// TIA Portal project "KananBagaliyev_Project" (V14)

(* hardware
DEVICE "S7300/ET200M station_1"  S7-300 station
   slot 0: "Rail_0"  Rail  6ES7 390-1***0-0AA0
   slot 1: "PS 307 10A_1"  PS 307 10A  6ES7 307-1KA02-0AA0
   slot 2: "PLC_1"  CPU 315-2 PN/DP  6ES7 315-2EH14-0AB0  V3.2
      slot 2: "PROFINET interface_1"  PN-IO
         slot 1: "Port_1"  Port
         slot 2: "Port_2"  Port
   slot 4: "DI 16x24VDC_1"  DI16 x 24VDC  6ES7 321-1BH50-0AA0
   slot 5: "DO 16x24VDC/0.5A_1"  DO16xDC24V/0.5A  6ES7 322-8BH10-0AB0
   slot 6: "AI 8x16BIT_1"  AI8 x 16 bits  6ES7 331-7NF10-0AB0
DEVICE "PC-System_1"  SIMATIC PC station
   slot 0: "SIMATIC PC station"  Rail  SIMATIC PC-Station  V1.0
      slot 125: "Stationmanager"  Station_Manager  V6.0.4
   slot 1: "HMI_RT_1"  WinCC RT Advanced  6AV2 104-0xxxx-xxxx  14.0.0.0
      slot 33792: "Host interface"  Host interface
   slot 2: "IE general_1"  IE General  IE_CP  V8.2.0
*)

// ===== PLC "PLC_1"  CPU 315-2 PN/DP =====

VAR_GLOBAL   // PLC tag table "Default tag table"
   "LT1401" AT %MW288 : Int;
   "LT1501" AT %MW290 : Int;
   "LT1601" AT %MW292 : Int;
   "LT1701" AT %MW294 : Int;
   "Pump100A_start" AT %M0.0 : Bool;
   "Pump100A_stop" AT %M0.1 : Bool;
   "Pump770A_start" AT %M0.2 : Bool;
   "Pump770A_stop" AT %M0.3 : Bool;
   "Pump771A_start" AT %M0.4 : Bool;
   "Pump771A_stop" AT %M0.5 : Bool;
   "Pump100A" AT %Q4.0 : Bool;
   "Pump770A" AT %Q4.1 : Bool;
   "Pump771A" AT %Q4.2 : Bool;
   "SV1401" AT %Q4.3 : Bool;
   "SV1402" AT %Q4.4 : Bool;
   "SV1501" AT %Q4.5 : Bool;
   "SV1502" AT %Q4.6 : Bool;
   "SV1601" AT %Q4.7 : Bool;
   "SV1602" AT %Q5.0 : Bool;
   "SV1701" AT %Q5.1 : Bool;
   "SV1702" AT %Q5.2 : Bool;
   "SV1401_open" AT %M0.6 : Bool;
   "SV1401_close" AT %M0.7 : Bool;
   "SV1402_open" AT %M1.0 : Bool;
   "SV1402_close" AT %M1.1 : Bool;
   "SV1501_open" AT %M1.2 : Bool;
   "SV1501_close" AT %M1.3 : Bool;
   "SV1502_open" AT %M1.4 : Bool;
   "SV1502_close" AT %M1.5 : Bool;
   "SV1601_open" AT %M1.6 : Bool;
   "SV1601_close" AT %M1.7 : Bool;
   "SV1602_open" AT %M2.0 : Bool;
   "SV1602_close" AT %M2.1 : Bool;
   "SV1701_open" AT %M2.2 : Bool;
   "SV1701_close" AT %M2.3 : Bool;
   "SV1702_open" AT %M2.4 : Bool;
   "SV1702_close" AT %M2.5 : Bool;
   "140L" AT %M2.6 : Bool;
   "140LL" AT %M2.7 : Bool;
   "140H" AT %M3.0 : Bool;
   "140HH" AT %M3.1 : Bool;
   "150L" AT %M3.2 : Bool;
   "150LL" AT %M3.3 : Bool;
   "150H" AT %M3.4 : Bool;
   "150HH" AT %M3.5 : Bool;
   "160L" AT %M3.6 : Bool;
   "160LL" AT %M3.7 : Bool;
   "160H" AT %M4.0 : Bool;
   "160HH" AT %M4.1 : Bool;
   "170L" AT %M4.2 : Bool;
   "170LL" AT %M4.3 : Bool;
   "170H" AT %M4.4 : Bool;
   "170HH" AT %M4.5 : Bool;
   "140_real" AT %MD200 : Real;
   "150_real" AT %MD204 : Real;
   "160_real" AT %MD208 : Real;
   "170_real" AT %MD212 : Real;
END_VAR

VAR_GLOBAL CONSTANT   // PLC tag table "Default tag table"
   "140L_SP" : Real := 150.0;
   "140LL_SP" : Real := 75.0;
   "140H_SP" : Real := 1350.0;
   "140HH_SP" : Real := 1425.0;
   "150L_SP" : Real := 250.0;
   "150LL_SP" : Real := 125.0;
   "150H_SP" : Real := 2250.0;
   "150HH_SP" : Real := 2375.0;
   "160L_SP" : Real := 300.0;
   "160LL_SP" : Real := 150.0;
   "160H_SP" : Real := 2700.0;
   "160HH_SP" : Real := 2850.0;
   "170L_SP" : Real := 1000.0;
   "170LL_SP" : Real := 500.0;
   "170H_SP" : Real := 9000.0;
   "170HH_SP" : Real := 9500.0;
   "140_capacity_max" : Real := 1500.0;
   "150_capacity_max" : Real := 2500.0;
   "160_capacity_max" : Real := 3000.0;
   "170_capacity_max" : Real := 10000.0;
   "140_capacity_min" : Real := 0.0;
   "150_capacity_min" : Real := 0.0;
   "160_capacity_min" : Real := 0.0;
   "170_capacity_min" : Real := 0.0;
END_VAR

DATA_BLOCK "FP_DB"   // DB1
{ S7_Optimized_Access := 'FALSE' }
VERSION : 0.1
   VAR
      FP_visibility_PUMP_100A : Bool := false;
      FP_visibility_PUMP_770A : Bool := false;
      FP_visibility_PUMP_771A : Bool := false;
      FP_tag_number_PUMP_100A : String := 'PUMP_100_A';
      FP_tag_number_PUMP_770A : String := 'PUMP_770_A';
      FP_tag_number_PUMP_771A : String := 'PUMP_771_A';
      FP_visibility_SV1401 : Bool := false;
      FP_visibility_SV1402 : Bool := false;
      FP_visibility_SV1501 : Bool := false;
      FP_visibility_SV1502 : Bool := false;
      FP_visibility_SV1601 : Bool := false;
      FP_visibility_SV1602 : Bool := false;
      FP_visibility_SV1701 : Bool := false;
      FP_visibility_SV1702 : Bool := false;
      FP_tag_number_SV1401 : String := 'SV1401';
      FP_tag_number_SV1402 : String := 'SV1402';
      FP_tag_number_SV1501 : String := 'SV1501';
      FP_tag_number_SV1502 : String := 'SV1502';
      FP_tag_number_SV1601 : String := 'SV1601';
      FP_tag_number_SV1602 : String := 'SV1602';
      FP_tag_number_SV1701 : String := 'SV1701';
      FP_tag_number_SV1702 : String := 'SV1702';
   END_VAR
BEGIN
END_DATA_BLOCK

DATA_BLOCK "Tank140Fill_DB"   // DB2
{ S7_Optimized_Access := 'FALSE' }
VERSION : 0.1
// stored: InstanceOfName FillTank
"FillTank"
BEGIN
END_DATA_BLOCK

DATA_BLOCK "Tank150Fill_DB"   // DB3
{ S7_Optimized_Access := 'FALSE' }
VERSION : 0.1
// stored: InstanceOfName FillTank
"FillTank"
BEGIN
END_DATA_BLOCK

DATA_BLOCK "Tank160Fill_DB"   // DB4
{ S7_Optimized_Access := 'FALSE' }
VERSION : 0.1
// stored: InstanceOfName FillTank
"FillTank"
BEGIN
END_DATA_BLOCK

DATA_BLOCK "DrainMasterTank_DB"   // DB5
{ S7_Optimized_Access := 'FALSE' }
VERSION : 0.1
// stored: InstanceOfName DrainMasterTank
"DrainMasterTank"
BEGIN
END_DATA_BLOCK

FUNCTION_BLOCK "FillTank"   // FB1, LAD
{ S7_Optimized_Access := 'FALSE' }
VERSION : 0.1
   VAR_INPUT
      SV1x02 : Bool;
      SV1x01 : Bool;
      Pump : Bool;
      Reduction_rate : Int;
   END_VAR
   VAR_IN_OUT
      LT1x01 : Int;
   END_VAR
   VAR
      "timer" : Time;
      IEC_Timer_0_Instance : TON;
      IEC_Timer_0_Instance_1 : TON;
      timer_1 : Time;
   END_VAR
BEGIN

REGION Network 1: Fill Tank timer
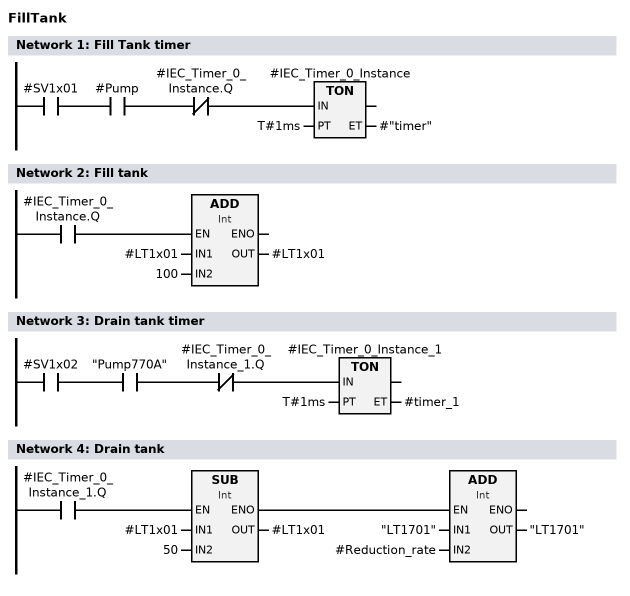
   #IEC_Timer_0_Instance.TON(IN := #SV1x01 AND #Pump AND NOT #IEC_Timer_0_Instance.Q,
                           PT := T#1ms,
                           ET => #"timer");
END_REGION

REGION Network 2: Fill tank
   RUNG wire#powerrail
      Contact( #IEC_Timer_0_Instance.Q )
      { S7_Templates := "SrcType := Int"; S7_GenerateENO := "TRUE" } Add(in1 := #LT1x01, in2 := 100, out => #LT1x01)
   END_RUNG
   // the same network as SCL:
   IF #IEC_Timer_0_Instance.Q THEN #LT1x01 := #LT1x01 + 100; END_IF;
END_REGION

REGION Network 3: Drain tank timer
   #IEC_Timer_0_Instance_1.TON(IN := #SV1x02 AND "Pump770A" AND NOT #IEC_Timer_0_Instance_1.Q,
                           PT := T#1ms,
                           ET => #timer_1);
END_REGION

REGION Network 4: Drain tank
   RUNG wire#powerrail
      Contact( #IEC_Timer_0_Instance_1.Q )
      { S7_Templates := "SrcType := Int"; S7_GenerateENO := "TRUE" } Sub(in1 := #LT1x01, in2 := 50, out => #LT1x01)
      { S7_Templates := "SrcType := Int"; S7_GenerateENO := "TRUE" } Add(in1 := "LT1701", in2 := #Reduction_rate, out => "LT1701")
   END_RUNG
   // the same network as SCL:
   // ENO of a box is taken as its EN; it also drops when the box reports an error
   IF #IEC_Timer_0_Instance_1.Q THEN
       #LT1x01 := #LT1x01 - 50;
       "LT1701" := "LT1701" + #Reduction_rate;
   END_IF;
END_REGION
END_FUNCTION_BLOCK

FUNCTION_BLOCK "DrainMasterTank"   // FB2, LAD
{ S7_Optimized_Access := 'FALSE' }
VERSION : 0.1
   VAR
      IEC_Timer_0_Instance : TON;
      "timer" : Time;
   END_VAR
BEGIN

REGION Network 1
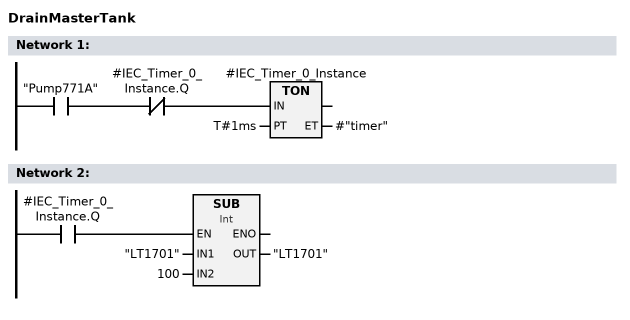
   #IEC_Timer_0_Instance.TON(IN := "Pump771A" AND NOT #IEC_Timer_0_Instance.Q, PT := T#1ms, ET => #"timer");
END_REGION

REGION Network 2
   RUNG wire#powerrail
      Contact( #IEC_Timer_0_Instance.Q )
      { S7_Templates := "SrcType := Int"; S7_GenerateENO := "TRUE" } Sub(in1 := "LT1701", in2 := 100, out => "LT1701")
   END_RUNG
   // the same network as SCL:
   IF #IEC_Timer_0_Instance.Q THEN "LT1701" := "LT1701" - 100; END_IF;
END_REGION
END_FUNCTION_BLOCK

FUNCTION "TankAlarm" : Void   // FC1, LAD
{ S7_Optimized_Access := 'FALSE' }
VERSION : 0.1
   VAR_INPUT
      LT1x01 : Int;
      max_level : Real;
      min_level : Real;
      high_alarm_sp : Real;
      low_alarm_sp : Real;
      hh_alarm_sp : Real;
      ll_alarm_sp : Real;
   END_VAR
   VAR_OUTPUT
      high_alarm : Bool;
      low_alarm : Bool;
      hh_alarm : Bool;
      ll_alarm : Bool;
   END_VAR
   VAR_IN_OUT
      level_real : Real;
   END_VAR
   VAR_TEMP
      bipolar : Bool;
      value : Word;
   END_VAR
BEGIN

REGION Network 1
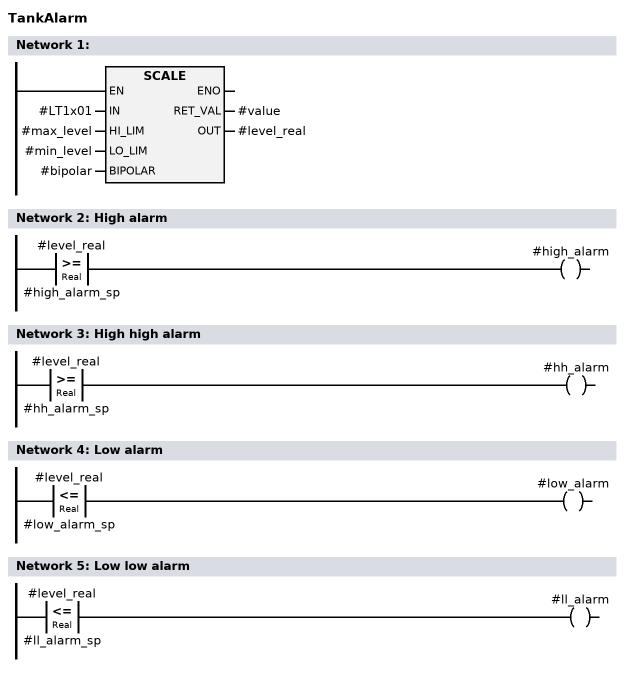
   #value := SCALE(IN := #LT1x01,
                   HI_LIM := #max_level,
                   LO_LIM := #min_level,
                   BIPOLAR := #bipolar,
                   OUT => #level_real);
END_REGION

REGION Network 2: High alarm
   RUNG wire#powerrail
      { S7_Templates := "SrcType := Real" } GE_Contact(in1 := #level_real, in2 := #high_alarm_sp)
      Coil( #high_alarm )
   END_RUNG
   // the same network as SCL:
   #high_alarm := #level_real >= #high_alarm_sp;
END_REGION

REGION Network 3: High high alarm
   RUNG wire#powerrail
      { S7_Templates := "SrcType := Real" } GE_Contact(in1 := #level_real, in2 := #hh_alarm_sp)
      Coil( #hh_alarm )
   END_RUNG
   // the same network as SCL:
   #hh_alarm := #level_real >= #hh_alarm_sp;
END_REGION

REGION Network 4: Low alarm
   RUNG wire#powerrail
      { S7_Templates := "SrcType := Real" } LE_Contact(in1 := #level_real, in2 := #low_alarm_sp)
      Coil( #low_alarm )
   END_RUNG
   // the same network as SCL:
   #low_alarm := #level_real <= #low_alarm_sp;
END_REGION

REGION Network 5: Low low alarm
   RUNG wire#powerrail
      { S7_Templates := "SrcType := Real" } LE_Contact(in1 := #level_real, in2 := #ll_alarm_sp)
      Coil( #ll_alarm )
   END_RUNG
   // the same network as SCL:
   #ll_alarm := #level_real <= #ll_alarm_sp;
END_REGION
END_FUNCTION

FUNCTION "SV1x01" : Void   // FC2, LAD
{ S7_Optimized_Access := 'FALSE' }
VERSION : 0.1
   VAR_INPUT
      Open_valve : Bool;
      Close_valve : Bool;
      HH_alarm : Bool;
      Inlet_pump_stop : Bool;
   END_VAR
   VAR_OUTPUT
      SV1x01 : Bool;
   END_VAR
BEGIN

REGION Network 1
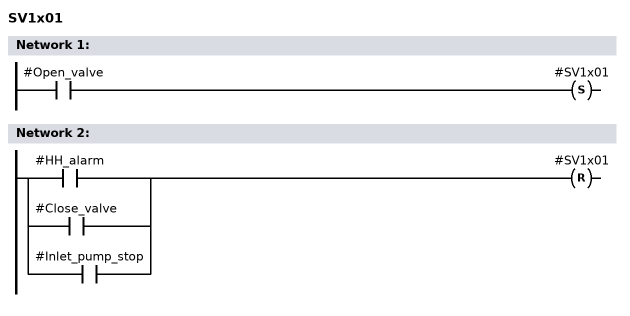
   RUNG wire#powerrail
      Contact( #Open_valve )
      S_Coil( #SV1x01 )
   END_RUNG
   // the same network as SCL:
   IF #Open_valve THEN #SV1x01 := TRUE; END_IF;
END_REGION

REGION Network 2
   RUNG wire#powerrail
      Contact( #HH_alarm )
      wire#w1
      R_Coil( #SV1x01 )
   END_RUNG
   RUNG wire#powerrail
      Contact( #Close_valve )
   END_RUNG wire#w1
   RUNG wire#powerrail
      Contact( #Inlet_pump_stop )
   END_RUNG wire#w1
   // the same network as SCL:
   IF #HH_alarm OR #Close_valve OR #Inlet_pump_stop THEN #SV1x01 := FALSE; END_IF;
END_REGION
END_FUNCTION

FUNCTION "Pump_100A" : Void   // FC3, LAD
{ S7_Optimized_Access := 'FALSE' }
VERSION : 0.1
   VAR_INPUT
      SV1x01_1 : Bool;
      SV1x01_2 : Bool;
      SV1x01_3 : Bool;
      Start_pump : Bool;
      Stop_pump : Bool;
   END_VAR
   VAR_OUTPUT
      Pump100A : Bool;
   END_VAR
BEGIN

REGION Network 1
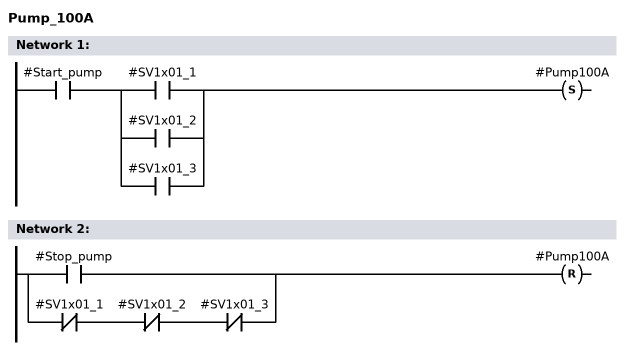
   RUNG wire#powerrail
      Contact( #Start_pump )
      wire#w1
      Contact( #SV1x01_1 )
      wire#w2
      S_Coil( #Pump100A )
   END_RUNG
   RUNG wire#w1
      Contact( #SV1x01_2 )
   END_RUNG wire#w2
   RUNG wire#w1
      Contact( #SV1x01_3 )
   END_RUNG wire#w2
   // the same network as SCL:
   IF #Start_pump AND (#SV1x01_1 OR #SV1x01_2 OR #SV1x01_3) THEN #Pump100A := TRUE; END_IF;
END_REGION

REGION Network 2
   RUNG wire#powerrail
      Contact( #Stop_pump )
      wire#w1
      R_Coil( #Pump100A )
   END_RUNG
   RUNG wire#powerrail
      I_Contact( #SV1x01_1 )
      I_Contact( #SV1x01_2 )
      I_Contact( #SV1x01_3 )
   END_RUNG wire#w1
   // the same network as SCL:
   IF #Stop_pump OR (NOT #SV1x01_1 AND NOT #SV1x01_2 AND NOT #SV1x01_3) THEN #Pump100A := FALSE; END_IF;
END_REGION
END_FUNCTION

FUNCTION "SV1x02_slaves" : Void   // FC4, LAD
{ S7_Optimized_Access := 'FALSE' }
VERSION : 0.1
   VAR_INPUT
      Valve_open : Bool;
      Valve_close : Bool;
      "170L" : Bool;
      "1x0L" : Bool;
      Pump_770_A_stop : Bool;
      "170H" : Bool;
   END_VAR
   VAR_OUTPUT
      Valve_energize : Bool;
   END_VAR
BEGIN

REGION Network 1
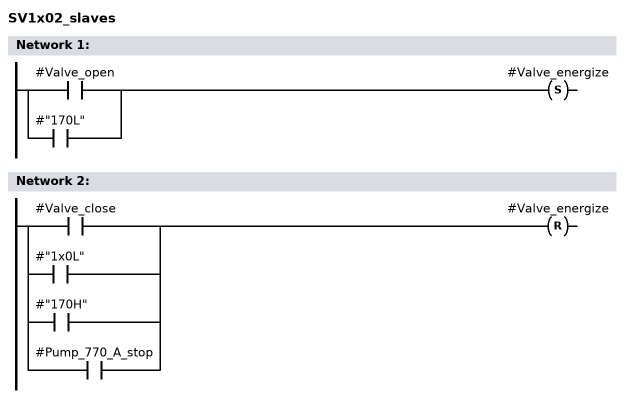
   RUNG wire#powerrail
      Contact( #Valve_open )
      wire#w1
      S_Coil( #Valve_energize )
   END_RUNG
   RUNG wire#powerrail
      Contact( #"170L" )
   END_RUNG wire#w1
   // the same network as SCL:
   IF #Valve_open OR #"170L" THEN #Valve_energize := TRUE; END_IF;
END_REGION

REGION Network 2
   RUNG wire#powerrail
      Contact( #Valve_close )
      wire#w1
      R_Coil( #Valve_energize )
   END_RUNG
   RUNG wire#powerrail
      Contact( #"1x0L" )
   END_RUNG wire#w1
   RUNG wire#powerrail
      Contact( #"170H" )
   END_RUNG wire#w1
   RUNG wire#powerrail
      Contact( #Pump_770_A_stop )
   END_RUNG wire#w1
   // the same network as SCL:
   IF #Valve_close OR #"1x0L" OR #"170H" OR #Pump_770_A_stop THEN #Valve_energize := FALSE; END_IF;
END_REGION
END_FUNCTION

FUNCTION "SV_1702" : Void   // FC5, LAD
{ S7_Optimized_Access := 'FALSE' }
VERSION : 0.1
   VAR_INPUT
      Valve_open : Bool;
      Valve_close : Bool;
      "170L" : Bool;
      Pump_771_A : Bool;
   END_VAR
   VAR_OUTPUT
      Valve_energize : Bool;
   END_VAR
BEGIN

REGION Network 1
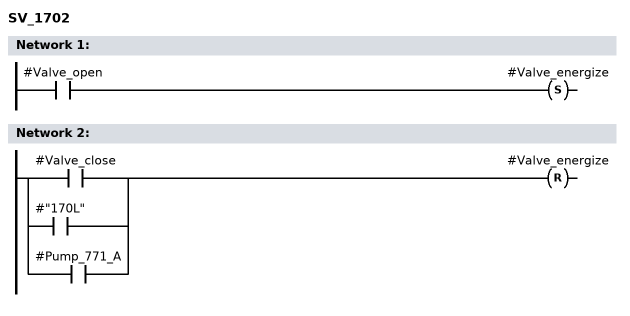
   RUNG wire#powerrail
      Contact( #Valve_open )
      S_Coil( #Valve_energize )
   END_RUNG
   // the same network as SCL:
   IF #Valve_open THEN #Valve_energize := TRUE; END_IF;
END_REGION

REGION Network 2
   RUNG wire#powerrail
      Contact( #Valve_close )
      wire#w1
      R_Coil( #Valve_energize )
   END_RUNG
   RUNG wire#powerrail
      Contact( #"170L" )
   END_RUNG wire#w1
   RUNG wire#powerrail
      Contact( #Pump_771_A )
   END_RUNG wire#w1
   // the same network as SCL:
   IF #Valve_close OR #"170L" OR #Pump_771_A THEN #Valve_energize := FALSE; END_IF;
END_REGION
END_FUNCTION

FUNCTION "Pump_770A" : Void   // FC6, LAD
{ S7_Optimized_Access := 'FALSE' }
VERSION : 0.1
   VAR_INPUT
      Start_pump : Bool;
      Stop_pump : Bool;
      SV1701 : Bool;
      SV1402 : Bool;
      SV1502 : Bool;
      SV1602 : Bool;
      "170L" : Bool;
      "170H" : Bool;
   END_VAR
   VAR_OUTPUT
      Pump_770A : Bool;
   END_VAR
BEGIN

REGION Network 1
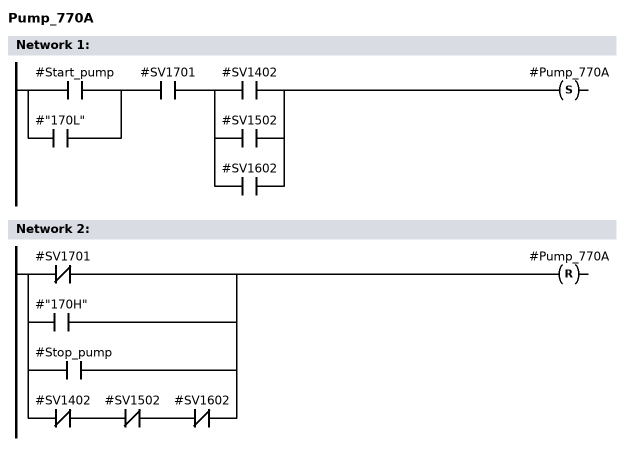
   RUNG wire#powerrail
      Contact( #Start_pump )
      wire#w1
      Contact( #SV1701 )
      wire#w2
      Contact( #SV1402 )
      wire#w3
      S_Coil( #Pump_770A )
   END_RUNG
   RUNG wire#powerrail
      Contact( #"170L" )
   END_RUNG wire#w1
   RUNG wire#w2
      Contact( #SV1502 )
   END_RUNG wire#w3
   RUNG wire#w2
      Contact( #SV1602 )
   END_RUNG wire#w3
   // the same network as SCL:
   IF (#Start_pump OR #"170L") AND #SV1701 AND (#SV1402 OR #SV1502 OR #SV1602) THEN
       #Pump_770A := TRUE;
   END_IF;
END_REGION

REGION Network 2
   RUNG wire#powerrail
      I_Contact( #SV1701 )
      wire#w1
      R_Coil( #Pump_770A )
   END_RUNG
   RUNG wire#powerrail
      Contact( #"170H" )
   END_RUNG wire#w1
   RUNG wire#powerrail
      Contact( #Stop_pump )
   END_RUNG wire#w1
   RUNG wire#powerrail
      I_Contact( #SV1402 )
      I_Contact( #SV1502 )
      I_Contact( #SV1602 )
   END_RUNG wire#w1
   // the same network as SCL:
   IF NOT #SV1701 OR #"170H" OR #Stop_pump OR (NOT #SV1402 AND NOT #SV1502 AND NOT #SV1602) THEN
       #Pump_770A := FALSE;
   END_IF;
END_REGION
END_FUNCTION

FUNCTION "Pump_771A" : Void   // FC7, LAD
{ S7_Optimized_Access := 'FALSE' }
VERSION : 0.1
   VAR_INPUT
      Pump_start : Bool;
      SV1702 : Bool;
      Pump_stop : Bool;
      "170L" : Bool;
   END_VAR
   VAR_OUTPUT
      Pump_771A : Bool;
   END_VAR
BEGIN

REGION Network 1
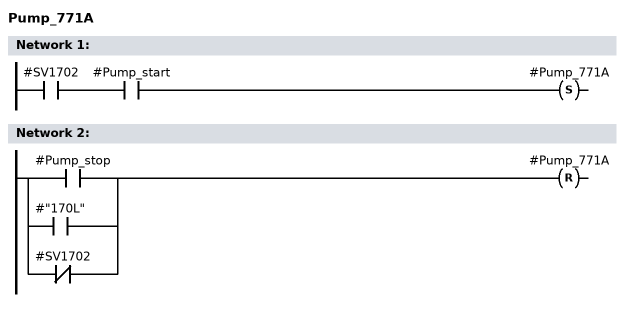
   RUNG wire#powerrail
      Contact( #SV1702 )
      Contact( #Pump_start )
      S_Coil( #Pump_771A )
   END_RUNG
   // the same network as SCL:
   IF #SV1702 AND #Pump_start THEN #Pump_771A := TRUE; END_IF;
END_REGION

REGION Network 2
   RUNG wire#powerrail
      Contact( #Pump_stop )
      wire#w1
      R_Coil( #Pump_771A )
   END_RUNG
   RUNG wire#powerrail
      Contact( #"170L" )
   END_RUNG wire#w1
   RUNG wire#powerrail
      I_Contact( #SV1702 )
   END_RUNG wire#w1
   // the same network as SCL:
   IF #Pump_stop OR #"170L" OR NOT #SV1702 THEN #Pump_771A := FALSE; END_IF;
END_REGION
END_FUNCTION

ORGANIZATION_BLOCK "Main"   // OB1, LAD
TITLE = "Main Program Sweep (Cycle)"
{ S7_Optimized_Access := 'FALSE' }
VERSION : 0.1
   VAR_TEMP
      OB1_EV_CLASS : Byte;   // Bits 0-3 = 1 (Coming event), Bits 4-7 = 1 (Event class 1)
      OB1_SCAN_1 : Byte;   // 1 (Cold restart scan 1 of OB 1), 3 (Scan 2-n of OB 1)
      OB1_PRIORITY : Byte;   // Priority of OB Execution
      OB1_OB_NUMBR : Byte;   // 1 (Organization block 1, OB1)
      OB1_RESERVED_1 : Byte;   // Reserved for system
      OB1_RESERVED_2 : Byte;   // Reserved for system
      OB1_PREV_CYCLE : Int;   // Cycle time of previous OB1 scan (milliseconds)
      OB1_MIN_CYCLE : Int;   // Minimum cycle time of OB1 (milliseconds)
      OB1_MAX_CYCLE : Int;   // Maximum cycle time of OB1 (milliseconds)
      OB1_DATE_TIME : Date_And_Time;   // Date and time OB1 started
   END_VAR
BEGIN

REGION Network 1: Tank 140
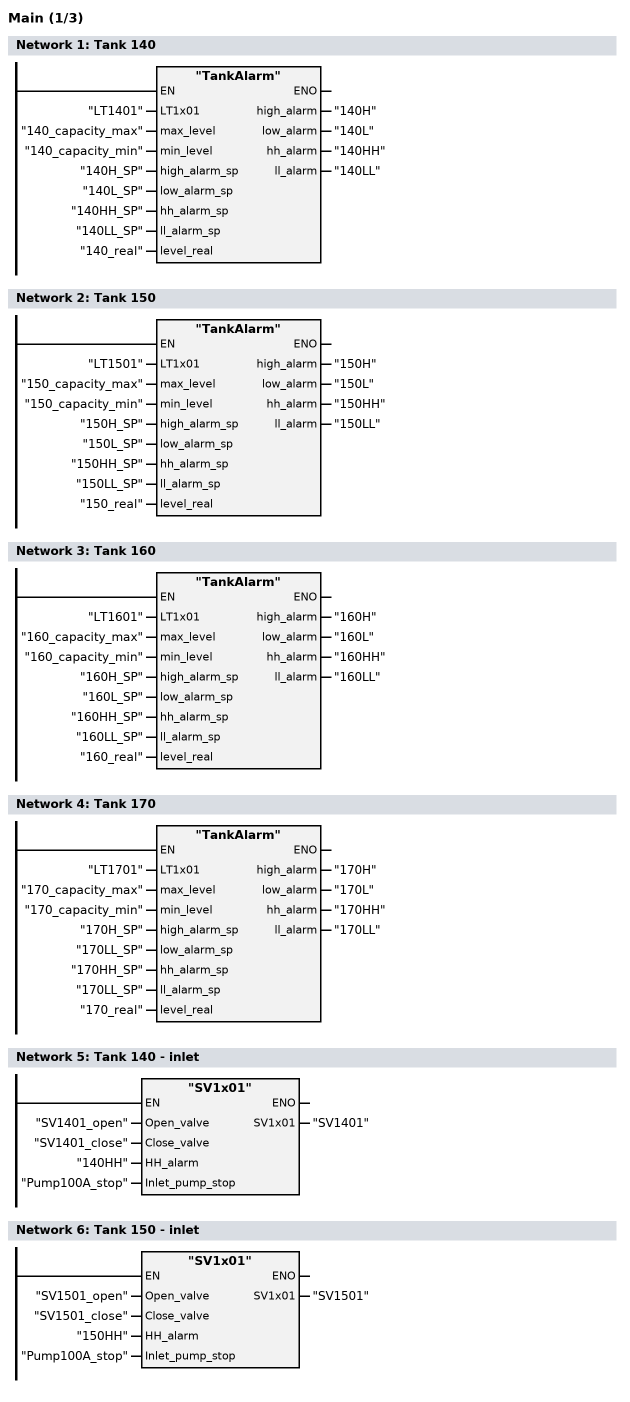
   RUNG wire#powerrail
      "TankAlarm"(LT1x01 := "LT1401", max_level := "140_capacity_max", min_level := "140_capacity_min", high_alarm_sp := "140H_SP", low_alarm_sp := "140L_SP", hh_alarm_sp := "140HH_SP", ll_alarm_sp := "140LL_SP", level_real := "140_real", high_alarm => "140H", low_alarm => "140L", hh_alarm => "140HH", ll_alarm => "140LL")
   END_RUNG
   // the same network as SCL:
   "TankAlarm"(LT1x01 := "LT1401",
               max_level := "140_capacity_max",
               min_level := "140_capacity_min",
               high_alarm_sp := "140H_SP",
               low_alarm_sp := "140L_SP",
               hh_alarm_sp := "140HH_SP",
               ll_alarm_sp := "140LL_SP",
               level_real := "140_real",
               high_alarm => "140H",
               low_alarm => "140L",
               hh_alarm => "140HH",
               ll_alarm => "140LL");
END_REGION

REGION Network 2: Tank 150
   RUNG wire#powerrail
      "TankAlarm"(LT1x01 := "LT1501", max_level := "150_capacity_max", min_level := "150_capacity_min", high_alarm_sp := "150H_SP", low_alarm_sp := "150L_SP", hh_alarm_sp := "150HH_SP", ll_alarm_sp := "150LL_SP", level_real := "150_real", high_alarm => "150H", low_alarm => "150L", hh_alarm => "150HH", ll_alarm => "150LL")
   END_RUNG
   // the same network as SCL:
   "TankAlarm"(LT1x01 := "LT1501",
               max_level := "150_capacity_max",
               min_level := "150_capacity_min",
               high_alarm_sp := "150H_SP",
               low_alarm_sp := "150L_SP",
               hh_alarm_sp := "150HH_SP",
               ll_alarm_sp := "150LL_SP",
               level_real := "150_real",
               high_alarm => "150H",
               low_alarm => "150L",
               hh_alarm => "150HH",
               ll_alarm => "150LL");
END_REGION

REGION Network 3: Tank 160
   RUNG wire#powerrail
      "TankAlarm"(LT1x01 := "LT1601", max_level := "160_capacity_max", min_level := "160_capacity_min", high_alarm_sp := "160H_SP", low_alarm_sp := "160L_SP", hh_alarm_sp := "160HH_SP", ll_alarm_sp := "160LL_SP", level_real := "160_real", high_alarm => "160H", low_alarm => "160L", hh_alarm => "160HH", ll_alarm => "160LL")
   END_RUNG
   // the same network as SCL:
   "TankAlarm"(LT1x01 := "LT1601",
               max_level := "160_capacity_max",
               min_level := "160_capacity_min",
               high_alarm_sp := "160H_SP",
               low_alarm_sp := "160L_SP",
               hh_alarm_sp := "160HH_SP",
               ll_alarm_sp := "160LL_SP",
               level_real := "160_real",
               high_alarm => "160H",
               low_alarm => "160L",
               hh_alarm => "160HH",
               ll_alarm => "160LL");
END_REGION

REGION Network 4: Tank 170
   RUNG wire#powerrail
      "TankAlarm"(LT1x01 := "LT1701", max_level := "170_capacity_max", min_level := "170_capacity_min", high_alarm_sp := "170H_SP", low_alarm_sp := "170LL_SP", hh_alarm_sp := "170HH_SP", ll_alarm_sp := "170LL_SP", level_real := "170_real", high_alarm => "170H", low_alarm => "170L", hh_alarm => "170HH", ll_alarm => "170LL")
   END_RUNG
   // the same network as SCL:
   "TankAlarm"(LT1x01 := "LT1701",
               max_level := "170_capacity_max",
               min_level := "170_capacity_min",
               high_alarm_sp := "170H_SP",
               low_alarm_sp := "170LL_SP",
               hh_alarm_sp := "170HH_SP",
               ll_alarm_sp := "170LL_SP",
               level_real := "170_real",
               high_alarm => "170H",
               low_alarm => "170L",
               hh_alarm => "170HH",
               ll_alarm => "170LL");
END_REGION

REGION Network 5: Tank 140 - inlet
   RUNG wire#powerrail
      "SV1x01"(Open_valve := "SV1401_open", Close_valve := "SV1401_close", HH_alarm := "140HH", Inlet_pump_stop := "Pump100A_stop", SV1x01 => "SV1401")
   END_RUNG
   // the same network as SCL:
   "SV1x01"(Open_valve := "SV1401_open",
            Close_valve := "SV1401_close",
            HH_alarm := "140HH",
            Inlet_pump_stop := "Pump100A_stop",
            SV1x01 => "SV1401");
END_REGION

REGION Network 6: Tank 150 - inlet
   RUNG wire#powerrail
      "SV1x01"(Open_valve := "SV1501_open", Close_valve := "SV1501_close", HH_alarm := "150HH", Inlet_pump_stop := "Pump100A_stop", SV1x01 => "SV1501")
   END_RUNG
   // the same network as SCL:
   "SV1x01"(Open_valve := "SV1501_open",
            Close_valve := "SV1501_close",
            HH_alarm := "150HH",
            Inlet_pump_stop := "Pump100A_stop",
            SV1x01 => "SV1501");
END_REGION

REGION Network 7: Tank 160 - inlet
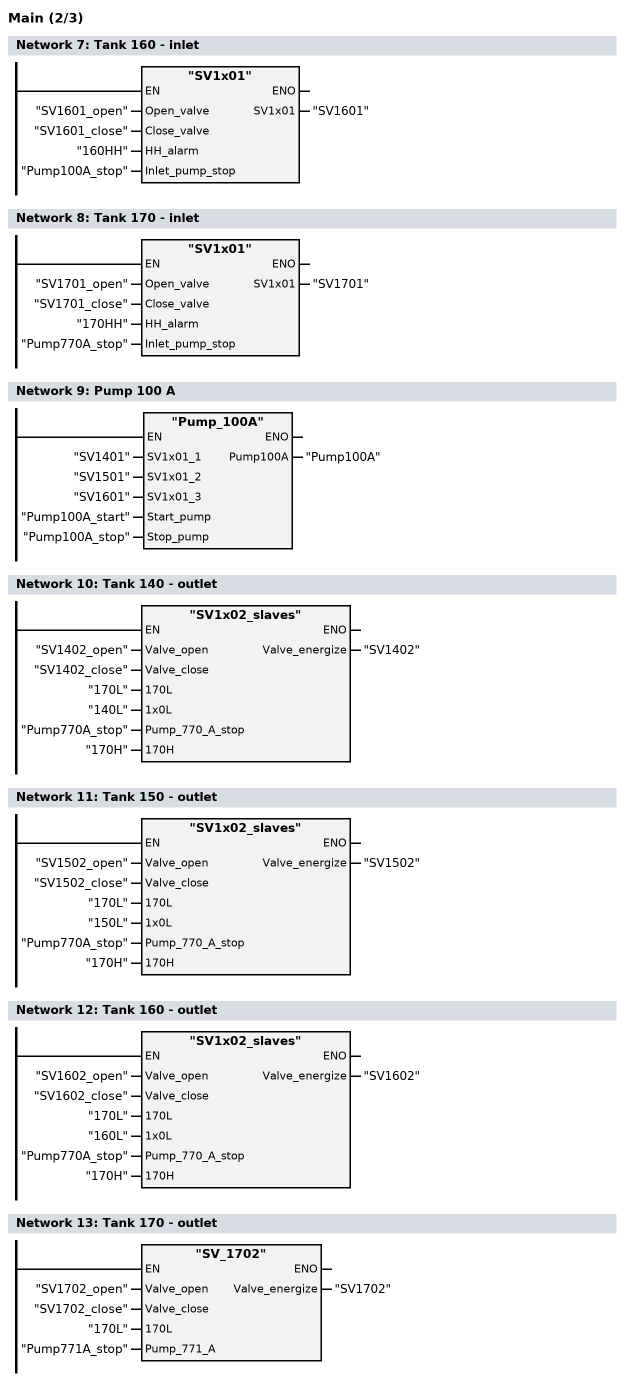
   RUNG wire#powerrail
      "SV1x01"(Open_valve := "SV1601_open", Close_valve := "SV1601_close", HH_alarm := "160HH", Inlet_pump_stop := "Pump100A_stop", SV1x01 => "SV1601")
   END_RUNG
   // the same network as SCL:
   "SV1x01"(Open_valve := "SV1601_open",
            Close_valve := "SV1601_close",
            HH_alarm := "160HH",
            Inlet_pump_stop := "Pump100A_stop",
            SV1x01 => "SV1601");
END_REGION

REGION Network 8: Tank 170 - inlet
   RUNG wire#powerrail
      "SV1x01"(Open_valve := "SV1701_open", Close_valve := "SV1701_close", HH_alarm := "170HH", Inlet_pump_stop := "Pump770A_stop", SV1x01 => "SV1701")
   END_RUNG
   // the same network as SCL:
   "SV1x01"(Open_valve := "SV1701_open",
            Close_valve := "SV1701_close",
            HH_alarm := "170HH",
            Inlet_pump_stop := "Pump770A_stop",
            SV1x01 => "SV1701");
END_REGION

REGION Network 9: Pump 100 A
   RUNG wire#powerrail
      "Pump_100A"(SV1x01_1 := "SV1401", SV1x01_2 := "SV1501", SV1x01_3 := "SV1601", Start_pump := "Pump100A_start", Stop_pump := "Pump100A_stop", Pump100A => "Pump100A")
   END_RUNG
   // the same network as SCL:
   "Pump_100A"(SV1x01_1 := "SV1401",
               SV1x01_2 := "SV1501",
               SV1x01_3 := "SV1601",
               Start_pump := "Pump100A_start",
               Stop_pump := "Pump100A_stop",
               Pump100A => "Pump100A");
END_REGION

REGION Network 10: Tank 140 - outlet
   RUNG wire#powerrail
      "SV1x02_slaves"(Valve_open := "SV1402_open", Valve_close := "SV1402_close", "170L" := "170L", "1x0L" := "140L", Pump_770_A_stop := "Pump770A_stop", "170H" := "170H", Valve_energize => "SV1402")
   END_RUNG
   // the same network as SCL:
   "SV1x02_slaves"(Valve_open := "SV1402_open",
                   Valve_close := "SV1402_close",
                   "170L" := "170L",
                   "1x0L" := "140L",
                   Pump_770_A_stop := "Pump770A_stop",
                   "170H" := "170H",
                   Valve_energize => "SV1402");
END_REGION

REGION Network 11: Tank 150 - outlet
   RUNG wire#powerrail
      "SV1x02_slaves"(Valve_open := "SV1502_open", Valve_close := "SV1502_close", "170L" := "170L", "1x0L" := "150L", Pump_770_A_stop := "Pump770A_stop", "170H" := "170H", Valve_energize => "SV1502")
   END_RUNG
   // the same network as SCL:
   "SV1x02_slaves"(Valve_open := "SV1502_open",
                   Valve_close := "SV1502_close",
                   "170L" := "170L",
                   "1x0L" := "150L",
                   Pump_770_A_stop := "Pump770A_stop",
                   "170H" := "170H",
                   Valve_energize => "SV1502");
END_REGION

REGION Network 12: Tank 160 - outlet
   RUNG wire#powerrail
      "SV1x02_slaves"(Valve_open := "SV1602_open", Valve_close := "SV1602_close", "170L" := "170L", "1x0L" := "160L", Pump_770_A_stop := "Pump770A_stop", "170H" := "170H", Valve_energize => "SV1602")
   END_RUNG
   // the same network as SCL:
   "SV1x02_slaves"(Valve_open := "SV1602_open",
                   Valve_close := "SV1602_close",
                   "170L" := "170L",
                   "1x0L" := "160L",
                   Pump_770_A_stop := "Pump770A_stop",
                   "170H" := "170H",
                   Valve_energize => "SV1602");
END_REGION

REGION Network 13: Tank 170 - outlet
   RUNG wire#powerrail
      "SV_1702"(Valve_open := "SV1702_open", Valve_close := "SV1702_close", "170L" := "170L", Pump_771_A := "Pump771A_stop", Valve_energize => "SV1702")
   END_RUNG
   // the same network as SCL:
   "SV_1702"(Valve_open := "SV1702_open",
             Valve_close := "SV1702_close",
             "170L" := "170L",
             Pump_771_A := "Pump771A_stop",
             Valve_energize => "SV1702");
END_REGION

REGION Network 14: Pump 770 A
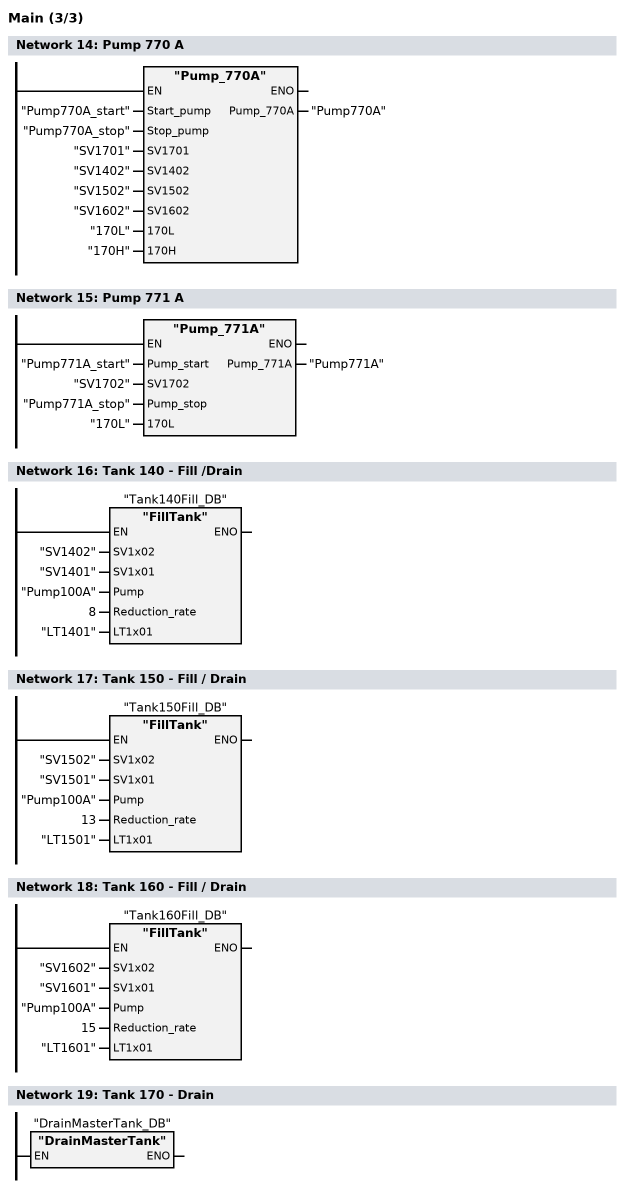
   RUNG wire#powerrail
      "Pump_770A"(Start_pump := "Pump770A_start", Stop_pump := "Pump770A_stop", SV1701 := "SV1701", SV1402 := "SV1402", SV1502 := "SV1502", SV1602 := "SV1602", "170L" := "170L", "170H" := "170H", Pump_770A => "Pump770A")
   END_RUNG
   // the same network as SCL:
   "Pump_770A"(Start_pump := "Pump770A_start",
               Stop_pump := "Pump770A_stop",
               SV1701 := "SV1701",
               SV1402 := "SV1402",
               SV1502 := "SV1502",
               SV1602 := "SV1602",
               "170L" := "170L",
               "170H" := "170H",
               Pump_770A => "Pump770A");
END_REGION

REGION Network 15: Pump 771 A
   RUNG wire#powerrail
      "Pump_771A"(Pump_start := "Pump771A_start", SV1702 := "SV1702", Pump_stop := "Pump771A_stop", "170L" := "170L", Pump_771A => "Pump771A")
   END_RUNG
   // the same network as SCL:
   "Pump_771A"(Pump_start := "Pump771A_start",
               SV1702 := "SV1702",
               Pump_stop := "Pump771A_stop",
               "170L" := "170L",
               Pump_771A => "Pump771A");
END_REGION

REGION Network 16: Tank 140 - Fill /Drain
   RUNG wire#powerrail
      "Tank140Fill_DB"(SV1x02 := "SV1402", SV1x01 := "SV1401", Pump := "Pump100A", Reduction_rate := 8, LT1x01 := "LT1401")
   END_RUNG
   // the same network as SCL:
   "Tank140Fill_DB"(SV1x02 := "SV1402",   // "FillTank"
                    SV1x01 := "SV1401",
                    Pump := "Pump100A",
                    Reduction_rate := 8,
                    LT1x01 := "LT1401");
END_REGION

REGION Network 17: Tank 150 - Fill / Drain
   RUNG wire#powerrail
      "Tank150Fill_DB"(SV1x02 := "SV1502", SV1x01 := "SV1501", Pump := "Pump100A", Reduction_rate := 13, LT1x01 := "LT1501")
   END_RUNG
   // the same network as SCL:
   "Tank150Fill_DB"(SV1x02 := "SV1502",   // "FillTank"
                    SV1x01 := "SV1501",
                    Pump := "Pump100A",
                    Reduction_rate := 13,
                    LT1x01 := "LT1501");
END_REGION

REGION Network 18: Tank 160 - Fill / Drain
   RUNG wire#powerrail
      "Tank160Fill_DB"(SV1x02 := "SV1602", SV1x01 := "SV1601", Pump := "Pump100A", Reduction_rate := 15, LT1x01 := "LT1601")
   END_RUNG
   // the same network as SCL:
   "Tank160Fill_DB"(SV1x02 := "SV1602",   // "FillTank"
                    SV1x01 := "SV1601",
                    Pump := "Pump100A",
                    Reduction_rate := 15,
                    LT1x01 := "LT1601");
END_REGION

REGION Network 19: Tank 170 - Drain
   RUNG wire#powerrail
      "DrainMasterTank_DB"()
   END_RUNG
   // the same network as SCL:
   "DrainMasterTank_DB"();   // "DrainMasterTank"
END_REGION
END_ORGANIZATION_BLOCK

(* ===== HMI "HMI_RT_1" =====
system functions are stored by id; their names below are inferred from use
connection "HMI_Connection_1": ETHERNET, SIMATIC S7 300/400 MPI

HMI tags "Default tag table"
   "140_real" : Real = PLC 140_real AT %MD200, 1 s
   "150_real" : Real = PLC 150_real AT %MD204, 1 s
   "160_real" : Real = PLC 160_real AT %MD208, 1 s
   "170_real" : Real = PLC 170_real AT %MD212, 1 s
   "Current_user" : WString[20], internal
   "Pump100A_start" : Bool = PLC Pump100A_start AT %M0.0, 1 s
   "Pump100A" : Bool = PLC Pump100A AT %Q4.0, 1 s
   "Pump100A_stop" : Bool = PLC Pump100A_stop AT %M0.1, 1 s
   "FP_DB_FP_visibility_PUMP_100A" : Bool = PLC FP_DB.FP_visibility_PUMP_100A AT %DB1.DBX0.0, 1 s
   "FP_DB_FP_tag_number_PUMP_100A" : String[254] = PLC FP_DB.FP_tag_number_PUMP_100A AT %DB1.DBX2.0, 1 s
   "140HH" : Bool = PLC 140HH AT %M3.1, 1 s
   "140LL" : Bool = PLC 140LL AT %M2.7, 1 s
   "150HH" : Bool = PLC 150HH AT %M3.5, 1 s
   "150LL" : Bool = PLC 150LL AT %M3.3, 1 s
   "160HH" : Bool = PLC 160HH AT %M4.1, 1 s
   "160L" : Bool = PLC 160L AT %M3.6, 1 s
   "160H" : Bool = PLC 160H AT %M4.0, 1 s
   "150L" : Bool = PLC 150L AT %M3.2, 1 s
   "150H" : Bool = PLC 150H AT %M3.4, 1 s
   "140L" : Bool = PLC 140L AT %M2.6, 1 s
   "140H" : Bool = PLC 140H AT %M3.0, 1 s
   "170H" : Bool = PLC 170H AT %M4.4, 1 s
   "170L" : Bool = PLC 170L AT %M4.2, 1 s
   "Pump770A" : Bool = PLC Pump770A AT %Q4.1, 1 s
   "Pump771A" : Bool = PLC Pump771A AT %Q4.2, 1 s
   "SV1401" : Bool = PLC SV1401 AT %Q4.3, 1 s
   "SV1402" : Bool = PLC SV1402 AT %Q4.4, 1 s
   "SV1501" : Bool = PLC SV1501 AT %Q4.5, 1 s
   "SV1502" : Bool = PLC SV1502 AT %Q4.6, 1 s
   "SV1601" : Bool = PLC SV1601 AT %Q4.7, 1 s
   "SV1602" : Bool = PLC SV1602 AT %Q5.0, 1 s
   "SV1701" : Bool = PLC SV1701 AT %Q5.1, 1 s
   "SV1702" : Bool = PLC SV1702 AT %Q5.2, 1 s
   "FP_DB_FP_visibility_SV1401" : Bool = PLC FP_DB.FP_visibility_SV1401 AT %DB1.DBX770.0, 1 s
   "SV1401_close" : Bool = PLC SV1401_close AT %M0.7, 1 s
   "SV1401_open" : Bool = PLC SV1401_open AT %M0.6, 1 s
   "FP_DB_FP_tag_number_SV1401" : String[254] = PLC FP_DB.FP_tag_number_SV1401 AT %DB1.DBX772.0, 1 s
   "FP_DB_FP_visibility_SV1402" : Bool = PLC FP_DB.FP_visibility_SV1402 AT %DB1.DBX770.1, 1 s
   "SV1402_close" : Bool = PLC SV1402_close AT %M1.1, 1 s
   "SV1402_open" : Bool = PLC SV1402_open AT %M1.0, 1 s
   "FP_DB_FP_tag_number_SV1402" : String[254] = PLC FP_DB.FP_tag_number_SV1402 AT %DB1.DBX1028.0, 1 s
   "FP_DB_FP_visibility_SV1501" : Bool = PLC FP_DB.FP_visibility_SV1501 AT %DB1.DBX770.2, 1 s
   "FP_DB_FP_visibility_SV1502" : Bool = PLC FP_DB.FP_visibility_SV1502 AT %DB1.DBX770.3, 1 s
   "FP_DB_FP_tag_number_SV1601" : String[254] = PLC FP_DB.FP_tag_number_SV1601 AT %DB1.DBX1796.0, 1 s
   "FP_DB_FP_visibility_SV1601" : Bool = PLC FP_DB.FP_visibility_SV1601 AT %DB1.DBX770.4, 1 s
   "FP_DB_FP_visibility_SV1602" : Bool = PLC FP_DB.FP_visibility_SV1602 AT %DB1.DBX770.5, 1 s
   "FP_DB_FP_visibility_SV1701" : Bool = PLC FP_DB.FP_visibility_SV1701 AT %DB1.DBX770.6, 1 s
   "FP_DB_FP_visibility_SV1702" : Bool = PLC FP_DB.FP_visibility_SV1702 AT %DB1.DBX770.7, 1 s
   "SV1501_close" : Bool = PLC SV1501_close AT %M1.3, 1 s
   "SV1501_open" : Bool = PLC SV1501_open AT %M1.2, 1 s
   "FP_DB_FP_tag_number_SV1501" : String[254] = PLC FP_DB.FP_tag_number_SV1501 AT %DB1.DBX1284.0, 1 s
   "SV1502_close" : Bool = PLC SV1502_close AT %M1.5, 1 s
   "SV1502_open" : Bool = PLC SV1502_open AT %M1.4, 1 s
   "FP_DB_FP_tag_number_SV1502" : String[254] = PLC FP_DB.FP_tag_number_SV1502 AT %DB1.DBX1540.0, 1 s
   "SV1601_close" : Bool = PLC SV1601_close AT %M1.7, 1 s
   "SV1601_open" : Bool = PLC SV1601_open AT %M1.6, 1 s
   "SV1602_close" : Bool = PLC SV1602_close AT %M2.1, 1 s
   "SV1602_open" : Bool = PLC SV1602_open AT %M2.0, 1 s
   "FP_DB_FP_tag_number_SV1602" : String[254] = PLC FP_DB.FP_tag_number_SV1602 AT %DB1.DBX2052.0, 1 s
   "SV1701_close" : Bool = PLC SV1701_close AT %M2.3, 1 s
   "SV1701_open" : Bool = PLC SV1701_open AT %M2.2, 1 s
   "FP_DB_FP_tag_number_SV1701" : String[254] = PLC FP_DB.FP_tag_number_SV1701 AT %DB1.DBX2308.0, 1 s
   "SV1702_close" : Bool = PLC SV1702_close AT %M2.5, 1 s
   "SV1702_open" : Bool = PLC SV1702_open AT %M2.4, 1 s
   "FP_DB_FP_tag_number_SV1702" : String[254] = PLC FP_DB.FP_tag_number_SV1702 AT %DB1.DBX2564.0, 1 s
   "FP_DB_FP_visibility_PUMP_770A" : Bool = PLC FP_DB.FP_visibility_PUMP_770A AT %DB1.DBX0.1, 1 s
   "Pump770A_start" : Bool = PLC Pump770A_start AT %M0.2, 1 s
   "Pump770A_stop" : Bool = PLC Pump770A_stop AT %M0.3, 1 s
   "FP_DB_FP_tag_number_PUMP_770A" : String[254] = PLC FP_DB.FP_tag_number_PUMP_770A AT %DB1.DBX258.0, 1 s
   "FP_DB_FP_visibility_PUMP_771A" : Bool = PLC FP_DB.FP_visibility_PUMP_771A AT %DB1.DBX0.2, 1 s
   "Pump771A_start" : Bool = PLC Pump771A_start AT %M0.4, 1 s
   "Pump771A_stop" : Bool = PLC Pump771A_stop AT %M0.5, 1 s
   "FP_DB_FP_tag_number_PUMP_771A" : String[254] = PLC FP_DB.FP_tag_number_PUMP_771A AT %DB1.DBX514.0, 1 s
   "LT1401" : Int = PLC LT1401 AT %MW288, 1 s

analog alarms
   1: 'Cause of alarm: High level in the tank Corrective action: Confirm that inlet SV is closed or outlet SV is opened in case of if Master tank is not in the high level, Pump 700A is running and SV1701 is open. Consequence of non action: Over pressure can cause explosion of the tank / High level of tank 140', class Acknowledgement, trigger "140_real"
   2: 'Cause of alarm: High level in the tank Corrective action: Confirm that inlet SV is closed or outlet SV is opened in case of if Master tank is not in the high level, Pump 700A is running and SV1701 is open. Consequence of non action: Over pressure can cause explosion of the tank / High level of tank 150', class Acknowledgement, trigger "150_real"
   3: 'High level of tank 160 / Cause of alarm: High level in the tank Corrective action: Confirm that inlet SV is closed or outlet SV is opened in case of if Master tank is not in the high level, Pump 700A is running and SV1701 is open. Consequence of non action: Over pressure can cause explosion of the tank', class Acknowledgement, trigger "160_real"
   4: 'High level of tank 170 / Cause of alarm: High level in the tank Corrective action: Confirm that inlet SV is closed or outlet SV is opened in case of if Master tank is not in the high level, Pump 700A is running and SV1701 is open. Consequence of non action: Over pressure can cause explosion of the tank', class Acknowledgement, trigger "170_real"
   5: 'Low level of tank 140 / Cause of alarm: Low level in the tank Corrective action: Confrim that inlet SV is opened or outlet SV is closed or Pump working. Consequence of non action: Pump will dry run', class Acknowledgement, trigger "140_real"
   6: 'Low level of tank 150 / Cause of alarm: Low level in the tank Corrective action: Confrim that inlet SV is opened or outlet SV is closed or Pump working. Consequence of non action: Pump will dry run', class Acknowledgement, trigger "150_real"
   7: 'Low level of tank 160 / Cause of alarm: Low level in the tank Corrective action: Confrim that inlet SV is opened or outlet SV is closed or Pump working. Consequence of non action: Pump will dry run', class Acknowledgement, trigger "160_real"
   8: 'Low level of tank 170 / Cause of alarm: Low level in the tank Corrective action: Confrim that inlet SV is opened or outlet SV is closed or Pump working. Also additionally be sure that outlet SVs of slave tanks are open. Consequence of non action: Pump will dry run', class Acknowledgement, trigger "170_real"

text list "Pump_status_list": 0 'Stopped'; 1 'Running'

screen "TankFarm" 1024x768
   Bar "Bar_4" at 351,490 size 70x129; MinimumValue 0; MaximumValue 10000
      ProcessValue <- "170_real"
   Bar "Bar_3" at 683,57 size 57x115; MinimumValue 0; MaximumValue 3000
      ProcessValue <- "160_real"
   Bar "Bar_2" at 417,60 size 57x115; MinimumValue 0; MaximumValue 2500
      ProcessValue <- "150_real"
   Bar "Bar_1" at 169,56 size 57x115; MinimumValue 0; MaximumValue 1500
      ProcessValue <- "140_real"
   GraphicView "Graphic view_4" at 227,161 size 24x172; Picture "Graphic_4"
   GraphicView "Graphic view_28" at 685,675 size 58x21; Picture "Graphic_10"
   GraphicView "Graphic view_26" at 561,674 size 95x21; Picture "Graphic_10"
   GraphicView "Graphic view_24" at 538,516 size 24x166; Picture "Graphic_4"
   GraphicView "Graphic view_21" at 450,518 size 24x166; Picture "Graphic_4"
   GraphicView "Graphic view_20" at 392,672 size 57x22; Picture "Graphic_10"
   GraphicView "Graphic view_7" at 485,161 size 24x166; Picture "Graphic_4"
   GraphicView "Graphic view_11" at 149,315 size 624x22; Picture "Graphic_10"
   GraphicView "Graphic view_8" at 818,161 size 24x266; Picture "Graphic_4"
   GraphicView "Graphic view_9" at 768,161 size 24x166; Picture "Graphic_4"
   GraphicView "Graphic view_6" at 535,161 size 24x281; Picture "Graphic_4"
   GraphicView "Graphic view_5" at 277,161 size 24x281; Picture "Graphic_4"
   GraphicView "Graphic view_10" at 124,315 size 52x50; Picture "Graphic_9"
   GraphicView "Graphic view_12" at 759,308 size 30x25; Picture "Graphic_11"
   GraphicView "Graphic view_13" at 811,415 size 27x24; Picture "Graphic_11"
   GraphicView "Graphic view_14" at 218,422 size 617x20; Picture "Graphic_10"
   GraphicView "Graphic view_16" at 216,426 size 27x24; Picture "Graphic_12"
   GraphicView "Graphic view_17" at 211,439 size 23x248; Picture "Graphic_4"
   GraphicView "Graphic view_19" at 216,677 size 27x24; Picture "Graphic_13"
   GraphicView "Graphic view_22" at 441,665 size 30x25; Picture "Graphic_11"
   GraphicView "Graphic view_23" at 725,661 size 52x50; Picture "Graphic_9"
   GraphicView "Graphic view_25" at 543,667 size 28x24; Picture "Graphic_13"
   GraphicView "Graphic view_27" at 651,655 size 44x40; Picture "Graphic_14"
   GraphicView "Graphic view_29" at 228,239 size 30x30; Picture "Graphic_16"
   GraphicView "Graphic view_30" at 277,239 size 30x30; Picture "Graphic_16"
   GraphicView "Graphic view_31" at 486,239 size 30x30; Picture "Graphic_16"
   GraphicView "Graphic view_32" at 535,239 size 30x30; Picture "Graphic_16"
   GraphicView "Graphic view_33" at 769,239 size 30x30; Picture "Graphic_16"
   GraphicView "Graphic view_34" at 818,239 size 30x30; Picture "Graphic_16"
   GraphicView "Graphic view_35" at 275,7 size 48x75; Picture "Graphic_17"
   GraphicView "Graphic view_1" at 216,38 size 107x141; Picture "Graphic_2"
   GraphicView "Graphic view_36" at 534,7 size 48x75; Picture "Graphic_17"
   GraphicView "Graphic view_37" at 834,7 size 48x75; Picture "Graphic_17"
   GraphicView "Graphic view_2" at 460,41 size 125x138; Picture "Graphic_2"
   GraphicView "Graphic view_3" at 727,38 size 151x141; Picture "Graphic_2"
   GraphicView "Graphic view_38" at 565,450 size 48x75; Picture "Graphic_17"
   GraphicView "Graphic view_15" at 403,471 size 210x156; Picture "Graphic_2"
   GraphicView "Graphic view_40" at 281,673 size 76x22; Picture "Graphic_10"
   GraphicView "Graphic view_18" at 234,672 size 52x50; Picture "Graphic_9"
   GraphicView "Graphic view_39" at 352,653 size 44x40; Picture "Graphic_14"
   Button "Button_1" at 231,86 size 79x26; TextOff 'Tank 140'; Authorization "Individual Tank Permission"
      on Click: ActivateScreen("Tank140", 0)
   Button "Button_2" at 485,85 size 79x26; TextOff 'Tank 150'; Authorization "Individual Tank Permission"
      on Click: ActivateScreen("Tank150", 0)
   Button "Button_3" at 767,86 size 79x26; TextOff 'Tank 160'; Authorization "Individual Tank Permission"
      on Click: ActivateScreen("Tank160", 0)
   Button "Button_4" at 474,516 size 79x26; TextOff 'Tank 170'; Authorization "Individual Tank Permission"
      on Click: ActivateScreen("Tank170", 0)
   Button "Button_5" at 878,717 size 134x39; TextOff 'Close Screen'
      on Click: StopRuntime(0)
   IOField "I/O field_1" at 176,9 size 96x32; FormatPattern 9999999
      ProcessValue <- "140_real"
   IOField "I/O field_2" at 431,9 size 96x32; FormatPattern 9999999
      ProcessValue <- "150_real"
   IOField "I/O field_3" at 725,6 size 96x32; FormatPattern 9999999
      ProcessValue <- "160_real"
   IOField "I/O field_4" at 374,443 size 96x32; FormatPattern 9999999
      ProcessValue <- "170_real"
   Button "Button_6" at 879,672 size 130x32; TextOff 'Main Page'
      on Press: ActivateScreen("LoginPage", 0)
   ScreenModuleView "FP_Pump_1" at 25,375 size 180x126; ScreenModuleType ""
      Guid_{11997190-7687} <- "Pump100A_start"
      Guid_{11997190-7691} <- "Pump100A"
      Guid_{11997190-7689} <- "Pump100A_stop"
      Guid_{11997190-7683} <- "FP_DB_FP_visibility_PUMP_100A"
      Guid_{11997190-7693} <- "FP_DB_FP_tag_number_PUMP_100A"
   Polygon "Polygon_1" at 311,147 size 22x21
      Visibility <- "140L"
   Polygon "Polygon_2" at 311,54 size 22x21
      Visibility <- "140H"
   Polygon "Polygon_3" at 571,147 size 22x21
      Visibility <- "150L"
   Polygon "Polygon_4" at 571,54 size 22x21
      Visibility <- "150H"
   Polygon "Polygon_5" at 869,147 size 22x21
      Visibility <- "160L"
   Polygon "Polygon_6" at 869,54 size 22x21
      Visibility <- "160H"
   Polygon "Polygon_7" at 601,590 size 22x21
      Visibility <- "170L"
   Polygon "Polygon_8" at 601,497 size 22x21
      Visibility <- "170H"
   Circle "Circle_1" at 134,327 size 23x23
      Appearance <- "Pump100A"
   Circle "Circle_2" at 245,685 size 23x23
      Appearance <- "Pump770A"
   Circle "Circle_3" at 735,673 size 23x23
      Appearance <- "Pump771A"
   Rectangle "Rectangle_1" at 280,244 size 19x18
      Appearance <- "SV1402"
   Rectangle "Rectangle_2" at 232,245 size 19x18
      Appearance <- "SV1401"
   Rectangle "Rectangle_3" at 490,245 size 19x18
      Appearance <- "SV1501"
   Rectangle "Rectangle_4" at 539,245 size 19x18
      Appearance <- "SV1502"
   Rectangle "Rectangle_5" at 773,245 size 19x18
      Appearance <- "SV1601"
   Rectangle "Rectangle_6" at 822,244 size 19x18
      Appearance <- "SV1602"
   Polygon "Polygon_9" at 357,654 size 34x13
      Appearance <- "SV1701"
   Polygon "Polygon_10" at 656,656 size 34x13
      Appearance <- "SV1702"
   Button "Button_7" at 121,308 size 55x59; TextOff 'Text'; Authorization "Operate"
      on Press: SetBit("FP_DB_FP_visibility_PUMP_100A")
   Button "Button_8" at 226,235 size 34x35; TextOff 'Text'; Authorization "Operate"
      on Press: SetBit("FP_DB_FP_visibility_SV1401"); ResetBit("FP_DB_FP_visibility_SV1402"); ResetBit("FP_DB_FP_visibility_SV1501"); ResetBit("FP_DB_FP_visibility_SV1502"); ResetBit("FP_DB_FP_visibility_SV1601"); ResetBit("FP_DB_FP_visibility_SV1602"); ResetBit("FP_DB_FP_visibility_SV1701"); ResetBit("FP_DB_FP_visibility_SV1702")
   ScreenModuleView "FP_Valve_1" at 28,175 size 180x143; ScreenModuleType ""
      Guid_{11997190-7683} <- "FP_DB_FP_visibility_SV1401"
      Guid_{11997190-7689} <- "SV1401_close"
      Guid_{11997190-7687} <- "SV1401_open"
      Guid_{11997190-7691} <- "SV1401"
      Guid_{11997190-7693} <- "FP_DB_FP_tag_number_SV1401"
   ScreenModuleView "FP_Valve_2" at 307,183 size 180x125; ScreenModuleType ""
      Guid_{11997190-7683} <- "FP_DB_FP_visibility_SV1402"
      Guid_{11997190-7689} <- "SV1402_close"
      Guid_{11997190-7687} <- "SV1402_open"
      Guid_{11997190-7691} <- "SV1402"
      Guid_{11997190-7693} <- "FP_DB_FP_tag_number_SV1402"
   Button "Button_9" at 272,236 size 34x35; TextOff 'Text'; Authorization "Operate"
      on Press: SetBit("FP_DB_FP_visibility_SV1402"); ResetBit("FP_DB_FP_visibility_SV1401"); ResetBit("FP_DB_FP_visibility_SV1501"); ResetBit("FP_DB_FP_visibility_SV1502"); ResetBit("FP_DB_FP_visibility_SV1601"); ResetBit("FP_DB_FP_visibility_SV1602"); ResetBit("FP_DB_FP_visibility_SV1701"); ResetBit("FP_DB_FP_visibility_SV1702")
   Button "Button_10" at 484,236 size 34x35; TextOff 'Text'; Authorization "Operate"
      on Press: SetBit("FP_DB_FP_visibility_SV1501"); ResetBit("FP_DB_FP_visibility_SV1402"); ResetBit("FP_DB_FP_visibility_SV1401"); ResetBit("FP_DB_FP_visibility_SV1502"); ResetBit("FP_DB_FP_visibility_SV1601"); ResetBit("FP_DB_FP_visibility_SV1602"); ResetBit("FP_DB_FP_visibility_SV1701"); ResetBit("FP_DB_FP_visibility_SV1702")
   Button "Button_11" at 533,235 size 34x35; TextOff 'Text'; Authorization "Operate"
      on Press: SetBit("FP_DB_FP_visibility_SV1502"); ResetBit("FP_DB_FP_visibility_SV1402"); ResetBit("FP_DB_FP_visibility_SV1501"); ResetBit("FP_DB_FP_visibility_SV1401"); ResetBit("FP_DB_FP_visibility_SV1601"); ResetBit("FP_DB_FP_visibility_SV1602"); ResetBit("FP_DB_FP_visibility_SV1701"); ResetBit("FP_DB_FP_visibility_SV1702")
   Button "Button_12" at 768,236 size 34x35; TextOff 'Text'; Authorization "Operate"
      on Press: SetBit("FP_DB_FP_visibility_SV1601"); ResetBit("FP_DB_FP_visibility_SV1402"); ResetBit("FP_DB_FP_visibility_SV1501"); ResetBit("FP_DB_FP_visibility_SV1502"); ResetBit("FP_DB_FP_visibility_SV1401"); ResetBit("FP_DB_FP_visibility_SV1602"); ResetBit("FP_DB_FP_visibility_SV1701"); ResetBit("FP_DB_FP_visibility_SV1702")
   Button "Button_13" at 817,236 size 34x35; TextOff 'Text'; Authorization "Operate"
      on Press: SetBit("FP_DB_FP_visibility_SV1602"); ResetBit("FP_DB_FP_visibility_SV1402"); ResetBit("FP_DB_FP_visibility_SV1501"); ResetBit("FP_DB_FP_visibility_SV1502"); ResetBit("FP_DB_FP_visibility_SV1601"); ResetBit("FP_DB_FP_visibility_SV1401"); ResetBit("FP_DB_FP_visibility_SV1701"); ResetBit("FP_DB_FP_visibility_SV1702")
   Button "Button_14" at 347,648 size 57x50; TextOff 'Text'; Authorization "Operate"
      on Press: SetBit("FP_DB_FP_visibility_SV1701"); ResetBit("FP_DB_FP_visibility_SV1402"); ResetBit("FP_DB_FP_visibility_SV1501"); ResetBit("FP_DB_FP_visibility_SV1502"); ResetBit("FP_DB_FP_visibility_SV1601"); ResetBit("FP_DB_FP_visibility_SV1602"); ResetBit("FP_DB_FP_visibility_SV1401"); ResetBit("FP_DB_FP_visibility_SV1702")
   Button "Button_15" at 645,650 size 57x50; TextOff 'Text'; Authorization "Operate"
      on Press: SetBit("FP_DB_FP_visibility_SV1702"); ResetBit("FP_DB_FP_visibility_SV1402"); ResetBit("FP_DB_FP_visibility_SV1501"); ResetBit("FP_DB_FP_visibility_SV1502"); ResetBit("FP_DB_FP_visibility_SV1601"); ResetBit("FP_DB_FP_visibility_SV1602"); ResetBit("FP_DB_FP_visibility_SV1701"); ResetBit("FP_DB_FP_visibility_SV1401")
   ScreenModuleView "FP_Valve_3" at 305,182 size 180x128; ScreenModuleType ""
      Guid_{11997190-7683} <- "FP_DB_FP_visibility_SV1501"
      Guid_{11997190-7687} <- "SV1501_open"
      Guid_{11997190-7691} <- "SV1501"
      Guid_{11997190-7693} <- "FP_DB_FP_tag_number_SV1501"
      Guid_{11997190-7689} <- "SV1501_close"
   ScreenModuleView "FP_Valve_4" at 584,182 size 180x132; ScreenModuleType ""
      Guid_{11997190-7683} <- "FP_DB_FP_visibility_SV1502"
      Guid_{11997190-7689} <- "SV1502_close"
      Guid_{11997190-7687} <- "SV1502_open"
      Guid_{11997190-7691} <- "SV1502"
      Guid_{11997190-7693} <- "FP_DB_FP_tag_number_SV1502"
   ScreenModuleView "FP_Valve_5" at 582,181 size 180x137; ScreenModuleType ""
      Guid_{11997190-7683} <- "FP_DB_FP_visibility_SV1601"
      Guid_{11997190-7687} <- "SV1601_open"
      Guid_{11997190-7691} <- "SV1601"
      Guid_{11997190-7693} <- "FP_DB_FP_tag_number_SV1601"
      Guid_{11997190-7689} <- "SV1601_close"
   ScreenModuleView "FP_Valve_6" at 842,182 size 180x128; ScreenModuleType ""
      Guid_{11997190-7683} <- "FP_DB_FP_visibility_SV1602"
      Guid_{11997190-7689} <- "SV1602_close"
      Guid_{11997190-7687} <- "SV1602_open"
      Guid_{11997190-7691} <- "SV1602"
      Guid_{11997190-7693} <- "FP_DB_FP_tag_number_SV1602"
   ScreenModuleView "FP_Valve_7" at 165,503 size 180x129; ScreenModuleType ""
      Guid_{11997190-7683} <- "FP_DB_FP_visibility_SV1701"
      Guid_{11997190-7689} <- "SV1701_close"
      Guid_{11997190-7687} <- "SV1701_open"
      Guid_{11997190-7691} <- "SV1701"
      Guid_{11997190-7693} <- "FP_DB_FP_tag_number_SV1701"
   ScreenModuleView "FP_Valve_8" at 634,516 size 180x126; ScreenModuleType ""
      Guid_{11997190-7683} <- "FP_DB_FP_visibility_SV1702"
      Guid_{11997190-7689} <- "SV1702_close"
      Guid_{11997190-7687} <- "SV1702_open"
      Guid_{11997190-7691} <- "SV1702"
      Guid_{11997190-7693} <- "FP_DB_FP_tag_number_SV1702"
   Button "Button_16" at 233,668 size 55x59; TextOff 'Text'; Authorization "Operate"
      on Press: SetBit("FP_DB_FP_visibility_PUMP_770A")
   ScreenModuleView "FP_Pump_2" at 16,632 size 180x127; ScreenModuleType ""
      Guid_{11997190-7683} <- "FP_DB_FP_visibility_PUMP_770A"
      Guid_{11997190-7687} <- "Pump770A_start"
      Guid_{11997190-7691} <- "Pump770A"
      Guid_{11997190-7689} <- "Pump770A_stop"
      Guid_{11997190-7693} <- "FP_DB_FP_tag_number_PUMP_770A"
   Button "Button_17" at 724,656 size 55x59; TextOff 'Text'; Authorization "Operate"
      on Press: SetBit("FP_DB_FP_visibility_PUMP_771A")
   ScreenModuleView "FP_Pump_3" at 818,503 size 180x129; ScreenModuleType ""
      Guid_{11997190-7683} <- "FP_DB_FP_visibility_PUMP_771A"
      Guid_{11997190-7687} <- "Pump771A_start"
      Guid_{11997190-7691} <- "Pump771A"
      Guid_{11997190-7689} <- "Pump771A_stop"
      Guid_{11997190-7693} <- "FP_DB_FP_tag_number_PUMP_771A"
   Button "Button_18" at 878,623 size 130x32; TextOff 'Alarm List'
      on Press: ActivateScreen("AlarmPage", 0)

Template "Tank1x0" 1024x768
   GraphicView "Template_Graphic view_13" at 44,18 size 87x81; Picture "Home"
   GraphicView "Template_Graphic view_4" at 172,229 size 131x22; Picture "Graphic_10"
   GraphicView "Template_Graphic view_2" at 115,229 size 74x52; Picture "Graphic_18"
   GraphicView "Template_Graphic view_3" at 333,229 size 131x22; Picture "Graphic_10"
   GraphicView "Template_Graphic view_5" at 291,219 size 53x37; Picture "Graphic_20"
   GraphicView "Template_Graphic view_6" at 558,360 size 22x67; Picture "Graphic_4"
   GraphicView "Template_Graphic view_8" at 580,421 size 131x22; Picture "Graphic_10"
   GraphicView "Template_Graphic view_10" at 734,421 size 131x22; Picture "Graphic_10"
   GraphicView "Template_Graphic view_9" at 697,411 size 53x37; Picture "Graphic_20"
   GraphicView "Template_Graphic view_7" at 562,413 size 27x26; Picture "Graphic_13"
   GraphicView "Template_Graphic view_11" at 852,405 size 74x52; Picture "Graphic_18"
   GraphicView "Template_Graphic view_12" at 553,150 size 41x90; Picture "Graphic_17"
   GraphicView "Template_Graphic view_1" at 437,183 size 161x213; Picture "Graphic_2"
   Button "Template_Button_1" at 44,18 size 87x80; TextOff 'Text'
      on Click: ActivateScreen("TankFarm", 0)

screen "Tank140" 1024x768, template "Tank1x0"
   IOField "I/O field_1" at 627,170 size 96x32; FormatPattern 9999999
      ProcessValue <- "140_real"
   Bar "Bar_1" at 627,210 size 70x180; MinimumValue 0; MaximumValue 1500
      ProcessValue <- "140_real"
   Polygon "Polygon_1" at 584,360 size 22x21
      Visibility <- "140L"
   Polygon "Polygon_2" at 584,215 size 22x21
      Visibility <- "140H"
   TextField "Text field_1" at 438,26 size 139x39; Text 'Tank 140'
   Button "Button_1" at 779,328 size 96x32; TextOff 'Tank 170'
      on Click: ActivateScreen("Tank170", 0)
   Button "Button_2" at 779,226 size 96x32; TextOff 'Tank 150'
      on Click: ActivateScreen("Tank150", 0)
   Button "Button_3" at 779,280 size 96x32; TextOff 'Tank 160'
      on Click: ActivateScreen("Tank160", 0)
   Rectangle "Rectangle_1" at 301,232 size 33x18
      Appearance <- "SV1401"
   Rectangle "Rectangle_2" at 707,424 size 33x18
      Appearance <- "SV1402"
   Button "Button_8" at 289,214 size 59x47; TextOff 'Text'
      on Press: SetBit("FP_DB_FP_visibility_SV1401"); ResetBit("FP_DB_FP_visibility_SV1402"); ResetBit("FP_DB_FP_visibility_SV1501"); ResetBit("FP_DB_FP_visibility_SV1502"); ResetBit("FP_DB_FP_visibility_SV1601"); ResetBit("FP_DB_FP_visibility_SV1602"); ResetBit("FP_DB_FP_visibility_SV1701"); ResetBit("FP_DB_FP_visibility_SV1702")
   Button "Button_9" at 694,407 size 57x45; TextOff 'Text'
      on Press: SetBit("FP_DB_FP_visibility_SV1402"); ResetBit("FP_DB_FP_visibility_SV1401"); ResetBit("FP_DB_FP_visibility_SV1501"); ResetBit("FP_DB_FP_visibility_SV1502"); ResetBit("FP_DB_FP_visibility_SV1601"); ResetBit("FP_DB_FP_visibility_SV1602"); ResetBit("FP_DB_FP_visibility_SV1701"); ResetBit("FP_DB_FP_visibility_SV1702")
   ScreenModuleView "FP_Valve_1" at 245,261 size 180x143; ScreenModuleType ""
      Guid_{11997190-7689} <- "SV1401_close"
      Guid_{11997190-7691} <- "SV1401"
      Guid_{11997190-7693} <- "FP_DB_FP_tag_number_SV1401"
      Guid_{11997190-7683} <- "FP_DB_FP_visibility_SV1401"
      Guid_{11997190-7687} <- "SV1401_open"
   ScreenModuleView "FP_Valve_2" at 648,452 size 180x125; ScreenModuleType ""
      Guid_{11997190-7689} <- "SV1402_close"
      Guid_{11997190-7691} <- "SV1402"
      Guid_{11997190-7693} <- "FP_DB_FP_tag_number_SV1402"
      Guid_{11997190-7683} <- "FP_DB_FP_visibility_SV1402"
      Guid_{11997190-7687} <- "SV1402_open"
   Circle "Circle_1" at 137,243 size 27x27
      Appearance <- "Pump100A"
   Button "Button_7" at 112,222 size 81x65; TextOff 'Text'
      on Press: SetBit("FP_DB_FP_visibility_PUMP_100A")
   ScreenModuleView "FP_Pump_1" at 54,287 size 180x144; ScreenModuleType ""
      Guid_{11997190-7689} <- "Pump100A_stop"
      Guid_{11997190-7691} <- "Pump100A"
      Guid_{11997190-7693} <- "FP_DB_FP_tag_number_PUMP_100A"
      Guid_{11997190-7683} <- "FP_DB_FP_visibility_PUMP_100A"
      Guid_{11997190-7687} <- "Pump100A_start"
   Circle "Circle_2" at 873,419 size 27x27
      Appearance <- "Pump770A"
   Button "Button_16" at 851,396 size 79x69; TextOff 'Text'
      on Press: SetBit("FP_DB_FP_visibility_PUMP_770A")
   ScreenModuleView "FP_Pump_2" at 842,465 size 180x144; ScreenModuleType ""
      Guid_{11997190-7689} <- "Pump770A_stop"
      Guid_{11997190-7691} <- "Pump770A"
      Guid_{11997190-7693} <- "FP_DB_FP_tag_number_PUMP_770A"
      Guid_{11997190-7683} <- "FP_DB_FP_visibility_PUMP_770A"
      Guid_{11997190-7687} <- "Pump770A_start"
   AlarmView "Alarm view_1" at 0,615 size 1023x153

screen "Tank150" 1024x768, template "Tank1x0"
   IOField "I/O field_1" at 627,170 size 96x32; FormatPattern 9999999
      ProcessValue <- "150_real"
   Bar "Bar_1" at 627,210 size 70x180; MinimumValue 0; MaximumValue 2500
      ProcessValue <- "150_real"
   Polygon "Polygon_3" at 584,360 size 22x21
      Visibility <- "150L"
   Polygon "Polygon_4" at 584,215 size 22x21
      Visibility <- "150H"
   TextField "Text field_1" at 438,26 size 139x39; Text 'Tank 150'
   Button "Button_1" at 779,226 size 96x32; TextOff 'Tank 140'
      on Click: ActivateScreen("Tank140", 0)
   Button "Button_2" at 779,280 size 96x32; TextOff 'Tank 160'
      on Click: ActivateScreen("Tank160", 0)
   Button "Button_3" at 779,328 size 96x32; TextOff 'Tank 170'
      on Click: ActivateScreen("Tank170", 0)
   Rectangle "Rectangle_1" at 301,232 size 33x18
      Appearance <- "SV1501"
   Rectangle "Rectangle_2" at 707,424 size 33x18
      Appearance <- "SV1502"
   Button "Button_10" at 288,212 size 60x49; TextOff 'Text'
      on Press: SetBit("FP_DB_FP_visibility_SV1501"); ResetBit("FP_DB_FP_visibility_SV1402"); ResetBit("FP_DB_FP_visibility_SV1401"); ResetBit("FP_DB_FP_visibility_SV1502"); ResetBit("FP_DB_FP_visibility_SV1601"); ResetBit("FP_DB_FP_visibility_SV1602"); ResetBit("FP_DB_FP_visibility_SV1701"); ResetBit("FP_DB_FP_visibility_SV1702")
   Button "Button_11" at 694,407 size 60x48; TextOff 'Text'
      on Press: SetBit("FP_DB_FP_visibility_SV1502"); ResetBit("FP_DB_FP_visibility_SV1402"); ResetBit("FP_DB_FP_visibility_SV1501"); ResetBit("FP_DB_FP_visibility_SV1401"); ResetBit("FP_DB_FP_visibility_SV1601"); ResetBit("FP_DB_FP_visibility_SV1602"); ResetBit("FP_DB_FP_visibility_SV1701"); ResetBit("FP_DB_FP_visibility_SV1702")
   ScreenModuleView "FP_Valve_3" at 236,269 size 180x128; ScreenModuleType ""
      Guid_{11997190-7689} <- "SV1501_close"
      Guid_{11997190-7691} <- "SV1501"
      Guid_{11997190-7693} <- "FP_DB_FP_tag_number_SV1501"
      Guid_{11997190-7683} <- "FP_DB_FP_visibility_SV1501"
      Guid_{11997190-7687} <- "SV1501_open"
   ScreenModuleView "FP_Valve_4" at 635,455 size 180x132; ScreenModuleType ""
      Guid_{11997190-7689} <- "SV1502_close"
      Guid_{11997190-7691} <- "SV1502"
      Guid_{11997190-7693} <- "FP_DB_FP_tag_number_SV1502"
      Guid_{11997190-7683} <- "FP_DB_FP_visibility_SV1502"
      Guid_{11997190-7687} <- "SV1502_open"
   Circle "Circle_1" at 137,243 size 27x27
      Appearance <- "Pump100A"
   Button "Button_7" at 112,222 size 81x65; TextOff 'Text'
      on Press: SetBit("FP_DB_FP_visibility_PUMP_100A")
   ScreenModuleView "FP_Pump_1" at 54,287 size 180x144; ScreenModuleType ""
      Guid_{11997190-7689} <- "Pump100A_stop"
      Guid_{11997190-7691} <- "Pump100A"
      Guid_{11997190-7693} <- "FP_DB_FP_tag_number_PUMP_100A"
      Guid_{11997190-7683} <- "FP_DB_FP_visibility_PUMP_100A"
      Guid_{11997190-7687} <- "Pump100A_start"
   Circle "Circle_2" at 873,419 size 27x27
      Appearance <- "Pump770A"
   Button "Button_16" at 851,396 size 79x69; TextOff 'Text'
      on Press: SetBit("FP_DB_FP_visibility_PUMP_770A")
   ScreenModuleView "FP_Pump_2" at 842,465 size 180x144; ScreenModuleType ""
      Guid_{11997190-7689} <- "Pump770A_stop"
      Guid_{11997190-7691} <- "Pump770A"
      Guid_{11997190-7693} <- "FP_DB_FP_tag_number_PUMP_770A"
      Guid_{11997190-7683} <- "FP_DB_FP_visibility_PUMP_770A"
      Guid_{11997190-7687} <- "Pump770A_start"
   AlarmView "Alarm view_1" at 0,615 size 1023x153

screen "Tank160" 1024x768, template "Tank1x0"
   IOField "I/O field_1" at 627,170 size 96x32; FormatPattern 9999999
      ProcessValue <- "160_real"
   Bar "Bar_1" at 627,210 size 70x180; MinimumValue 0; MaximumValue 3000
      ProcessValue <- "160_real"
   Polygon "Polygon_5" at 584,360 size 22x21
      Visibility <- "160L"
   Polygon "Polygon_6" at 584,215 size 22x21
      Visibility <- "160H"
   TextField "Text field_1" at 438,26 size 139x39; Text 'Tank 160'
   Button "Button_1" at 779,226 size 96x32; TextOff 'Tank 140'
      on Click: ActivateScreen("Tank140", 0)
   Button "Button_2" at 779,280 size 96x32; TextOff 'Tank 150'
      on Click: ActivateScreen("Tank150", 0)
   Button "Button_3" at 779,328 size 96x32; TextOff 'Tank 170'
      on Click: ActivateScreen("Tank170", 0)
   Rectangle "Rectangle_2" at 707,424 size 33x18
      Appearance <- "SV1602"
   Rectangle "Rectangle_1" at 301,232 size 33x18
      Appearance <- "SV1601"
   Button "Button_12" at 288,215 size 61x43; TextOff 'Text'
      on Press: SetBit("FP_DB_FP_visibility_SV1601"); ResetBit("FP_DB_FP_visibility_SV1402"); ResetBit("FP_DB_FP_visibility_SV1501"); ResetBit("FP_DB_FP_visibility_SV1502"); ResetBit("FP_DB_FP_visibility_SV1401"); ResetBit("FP_DB_FP_visibility_SV1602"); ResetBit("FP_DB_FP_visibility_SV1701"); ResetBit("FP_DB_FP_visibility_SV1702")
   Button "Button_13" at 695,408 size 57x43; TextOff 'Text'
      on Press: SetBit("FP_DB_FP_visibility_SV1602"); ResetBit("FP_DB_FP_visibility_SV1402"); ResetBit("FP_DB_FP_visibility_SV1501"); ResetBit("FP_DB_FP_visibility_SV1502"); ResetBit("FP_DB_FP_visibility_SV1601"); ResetBit("FP_DB_FP_visibility_SV1401"); ResetBit("FP_DB_FP_visibility_SV1701"); ResetBit("FP_DB_FP_visibility_SV1702")
   ScreenModuleView "FP_Valve_5" at 240,257 size 180x137; ScreenModuleType ""
      Guid_{11997190-7689} <- "SV1601_close"
      Guid_{11997190-7691} <- "SV1601"
      Guid_{11997190-7693} <- "FP_DB_FP_tag_number_SV1601"
      Guid_{11997190-7683} <- "FP_DB_FP_visibility_SV1601"
      Guid_{11997190-7687} <- "SV1601_open"
   ScreenModuleView "FP_Valve_6" at 642,458 size 180x128; ScreenModuleType ""
      Guid_{11997190-7689} <- "SV1602_close"
      Guid_{11997190-7691} <- "SV1602"
      Guid_{11997190-7693} <- "FP_DB_FP_tag_number_SV1602"
      Guid_{11997190-7683} <- "FP_DB_FP_visibility_SV1602"
      Guid_{11997190-7687} <- "SV1602_open"
   Circle "Circle_1" at 137,243 size 27x27
      Appearance <- "Pump100A"
   Button "Button_7" at 112,222 size 81x65; TextOff 'Text'
      on Press: SetBit("FP_DB_FP_visibility_PUMP_100A")
   ScreenModuleView "FP_Pump_1" at 54,287 size 180x144; ScreenModuleType ""
      Guid_{11997190-7689} <- "Pump100A_stop"
      Guid_{11997190-7691} <- "Pump100A"
      Guid_{11997190-7693} <- "FP_DB_FP_tag_number_PUMP_100A"
      Guid_{11997190-7683} <- "FP_DB_FP_visibility_PUMP_100A"
      Guid_{11997190-7687} <- "Pump100A_start"
   Circle "Circle_2" at 873,419 size 27x27
      Appearance <- "Pump770A"
   Button "Button_16" at 851,396 size 79x69; TextOff 'Text'
      on Press: SetBit("FP_DB_FP_visibility_PUMP_770A")
   ScreenModuleView "FP_Pump_2" at 842,465 size 180x144; ScreenModuleType ""
      Guid_{11997190-7689} <- "Pump770A_stop"
      Guid_{11997190-7691} <- "Pump770A"
      Guid_{11997190-7693} <- "FP_DB_FP_tag_number_PUMP_770A"
      Guid_{11997190-7683} <- "FP_DB_FP_visibility_PUMP_770A"
      Guid_{11997190-7687} <- "Pump770A_start"
   AlarmView "Alarm view_1" at 0,615 size 1023x153

screen "Tank170" 1024x768, template "Tank1x0"
   IOField "I/O field_4" at 627,170 size 96x32; FormatPattern 9999999
      ProcessValue <- "170_real"
   Bar "Bar_4" at 627,210 size 70x180; MinimumValue 0; MaximumValue 10000
      ProcessValue <- "170_real"
   Polygon "Polygon_7" at 584,360 size 22x21
      Visibility <- "170L"
   Polygon "Polygon_8" at 584,215 size 22x21
      Visibility <- "170H"
   TextField "Text field_1" at 438,26 size 139x39; Text 'Tank 170'
   Button "Button_1" at 779,226 size 96x32; TextOff 'Tank 140'
      on Click: ActivateScreen("Tank140", 0)
   Button "Button_2" at 779,280 size 96x32; TextOff 'Tank 150'
      on Click: ActivateScreen("Tank150", 0)
   Button "Button_3" at 779,328 size 96x32; TextOff 'Tank 160'
      on Click: ActivateScreen("Tank160", 0)
   Rectangle "Rectangle_2" at 707,424 size 33x18
      Appearance <- "SV1702"
   Rectangle "Rectangle_1" at 301,232 size 33x18
      Appearance <- "SV1701"
   Button "Button_14" at 290,210 size 57x50; TextOff 'Text'
      on Press: SetBit("FP_DB_FP_visibility_SV1701"); ResetBit("FP_DB_FP_visibility_SV1402"); ResetBit("FP_DB_FP_visibility_SV1501"); ResetBit("FP_DB_FP_visibility_SV1502"); ResetBit("FP_DB_FP_visibility_SV1601"); ResetBit("FP_DB_FP_visibility_SV1602"); ResetBit("FP_DB_FP_visibility_SV1401"); ResetBit("FP_DB_FP_visibility_SV1702")
   Button "Button_15" at 696,405 size 57x50; TextOff 'Text'
      on Press: SetBit("FP_DB_FP_visibility_SV1702"); ResetBit("FP_DB_FP_visibility_SV1402"); ResetBit("FP_DB_FP_visibility_SV1501"); ResetBit("FP_DB_FP_visibility_SV1502"); ResetBit("FP_DB_FP_visibility_SV1601"); ResetBit("FP_DB_FP_visibility_SV1602"); ResetBit("FP_DB_FP_visibility_SV1701"); ResetBit("FP_DB_FP_visibility_SV1401")
   ScreenModuleView "FP_Valve_7" at 244,272 size 180x129; ScreenModuleType ""
      Guid_{11997190-7689} <- "SV1701_close"
      Guid_{11997190-7691} <- "SV1701"
      Guid_{11997190-7693} <- "FP_DB_FP_tag_number_SV1701"
      Guid_{11997190-7683} <- "FP_DB_FP_visibility_SV1701"
      Guid_{11997190-7687} <- "SV1701_open"
   ScreenModuleView "FP_Valve_8" at 637,461 size 180x126; ScreenModuleType ""
      Guid_{11997190-7689} <- "SV1702_close"
      Guid_{11997190-7691} <- "SV1702"
      Guid_{11997190-7693} <- "FP_DB_FP_tag_number_SV1702"
      Guid_{11997190-7683} <- "FP_DB_FP_visibility_SV1702"
      Guid_{11997190-7687} <- "SV1702_open"
   Circle "Circle_1" at 137,243 size 27x27
      Appearance <- "Pump770A"
   Button "Button_7" at 112,222 size 81x65; TextOff 'Text'
      on Press: SetBit("FP_DB_FP_visibility_PUMP_770A")
   ScreenModuleView "FP_Pump_3" at 54,287 size 180x144; ScreenModuleType ""
      Guid_{11997190-7689} <- "Pump771A_stop"
      Guid_{11997190-7691} <- "Pump771A"
      Guid_{11997190-7693} <- "FP_DB_FP_tag_number_PUMP_771A"
      Guid_{11997190-7683} <- "FP_DB_FP_visibility_PUMP_771A"
      Guid_{11997190-7687} <- "Pump771A_start"
   Circle "Circle_2" at 873,419 size 27x27
      Appearance <- "Pump771A"
   Button "Button_16" at 851,400 size 79x69; TextOff 'Text'
      on Press: SetBit("FP_DB_FP_visibility_PUMP_771A")
   ScreenModuleView "FP_Pump_2" at 842,465 size 180x144; ScreenModuleType ""
      Guid_{11997190-7689} <- "Pump770A_stop"
      Guid_{11997190-7691} <- "Pump770A"
      Guid_{11997190-7693} <- "FP_DB_FP_tag_number_PUMP_770A"
      Guid_{11997190-7683} <- "FP_DB_FP_visibility_PUMP_770A"
      Guid_{11997190-7687} <- "Pump770A_start"
   AlarmView "Alarm view_1" at 0,615 size 1023x153

screen "LoginPage" 1024x768
   Button "Button_1" at 247,49 size 96x32; TextOff 'LogIn'
      on Press: function_a2a04561()
   Button "Button_2" at 368,49 size 96x32; TextOff 'Log out'
      on Press: function_f23ef4c9()
   Button "Button_3" at 397,139 size 288x56; TextOff 'Tank Farm'; Authorization "Authorization"
      on Press: ActivateScreen("TankFarm", 0)
   IOField "I/O field_1" at 669,49 size 219x32; FormatPattern ????????????????????
      ProcessValue <- "Current_user"
   TextField "Text field_1" at 552,53 size 101x22; Text 'Current User'
   UserView "User view_1" at 101,254 size 821x240
   GraphicView "Graphic view_1" at 939,0 size 85x57; Picture "Graphic_22"

Template "SlavePumps" 1024x768
   Circle "Circle_1" at 137,243 size 27x27
      Appearance <- "Pump100A"
   Button "Button_7" at 112,222 size 81x65; TextOff 'Text'
      on Press: SetBit("FP_DB_FP_visibility_PUMP_100A")
   ScreenModuleView "FP_Pump_1" at 54,287 size 180x254; ScreenModuleType ""
      Guid_{11997190-7689} <- "Pump100A_stop"
      Guid_{11997190-7691} <- "Pump100A"
      Guid_{11997190-7693} <- "FP_DB_FP_tag_number_PUMP_100A"
      Guid_{11997190-7683} <- "FP_DB_FP_visibility_PUMP_100A"
      Guid_{11997190-7687} <- "Pump100A_start"
   ScreenModuleView "FP_Pump_3" at 793,137 size 180x254; ScreenModuleType ""
      Guid_{11997190-7689} <- "Pump771A_stop"
      Guid_{11997190-7691} <- "Pump771A"
      Guid_{11997190-7693} <- "FP_DB_FP_tag_number_PUMP_771A"
      Guid_{11997190-7683} <- "FP_DB_FP_visibility_PUMP_771A"
      Guid_{11997190-7687} <- "Pump771A_start"
   Circle "Circle_2" at 873,419 size 27x27
      Appearance <- "Pump770A"
   Button "Button_16" at 851,396 size 79x69; TextOff 'Text'
      on Press: SetBit("FP_DB_FP_visibility_PUMP_770A")

screen "AlarmPage" 1024x768
   AlarmView "Alarm view_1" at 0,126 size 1023x641; Authorization "Operate"
   TextField "Text field_1" at 292,25 size 351x91; Text 'Alarm list'
   GraphicView "Template_Graphic view_13" at 44,18 size 87x81; Picture "Home"
   Button "Template_Button_1" at 44,18 size 87x80; TextOff 'Text'
      on Click: ActivateScreen("TankFarm", 0)

scheduled task "User_change"
   on Action: function_f41c6f6c("Current_user")
*)

(* ===== HMI "HMI_RT_1" =====
system functions are stored by id; their names below are inferred from use

text list "Pump_status_list": 0 'Stopped'; 1 'Running'

text list "Valve_status_list": 0 'Closed'; 1 'Opened'

ScreenModuleEditorView "FP_Valve" 640x480
   Rectangle "Rectangle_1" at 246,32 size 153x141
      Visibility <- "FP_visibility"
   Button "Button_7" at 362,53 size 27x26; TextOff 'X'
      on Press: ResetBit("FP_visibility")
      Visibility <- "FP_visibility"
   Button "Button_8" at 254,135 size 60x24; TextOff 'Open'
      on Press: function_b14e0dd5("Valve_open", 0)
      Visibility <- "FP_visibility"
   Button "Button_9" at 320,134 size 69x25; TextOff 'Close'
      on Press: function_b14e0dd5("Valve_close", 0)
      Visibility <- "FP_visibility"
   IOField "I/O field_5" at 254,47 size 91x32; FormatPattern ??????????
      ProcessValue <- "Valve_tag_number"
      Visibility <- "FP_visibility"
   SymbolicIOField "Symbolic I/O field_1" at 315,91 size 74x32; TextOn '1'; TextOff '0'; TextList "Valve_status_list"
      ProcessValue <- "Valve_status"
      Visibility <- "FP_visibility"
   TextField "Text field_1" at 256,96 size 53x22; Text 'Status'
      Visibility <- "FP_visibility"
*)

(* ===== HMI "HMI_RT_1" =====
system functions are stored by id; their names below are inferred from use

text list "Pump_status_list": 0 'Stopped'; 1 'Running'

ScreenModuleEditorView "FP_Pump" 640x480
   Rectangle "Rectangle_1" at 219,32 size 180x158
      Visibility <- "FP_visibility"
   Button "Button_7" at 362,40 size 27x38; TextOff 'X'
      on Press: ResetBit("FP_visibility")
      Visibility <- "FP_visibility"
   Button "Button_8" at 229,139 size 67x32; TextOff 'Start'
      on Press: function_b14e0dd5("Pump_start", 0)
      Visibility <- "FP_visibility"
   Button "Button_9" at 322,139 size 67x32; TextOff 'Stop'
      on Press: function_b14e0dd5("Pump_stop", 0)
      Visibility <- "FP_visibility"
   IOField "I/O field_5" at 229,46 size 128x32; FormatPattern ??????????
      ProcessValue <- "Pump_tag_number"
      Visibility <- "FP_visibility"
   SymbolicIOField "Symbolic I/O field_1" at 293,95 size 96x32; TextOn '1'; TextOff '0'; TextList "Pump_status_list"
      ProcessValue <- "Pump_status"
      Visibility <- "FP_visibility"
   TextField "Text field_1" at 229,94 size 53x22; Text 'Status'
      Visibility <- "FP_visibility"
*)